C03563=1012.547,271.905,-142.723,165.559,65.313,161.899
C03564=1012.520,272.316,-142.820,165.483,65.289,161.863
C03565=1012.492,272.726,-142.918,165.407,65.263,161.827
C03566=1012.478,272.932,-142.967,165.366,65.262,161.811
C03567=1012.464,273.137,-143.018,165.328,65.252,161.794
C03568=1012.450,273.343,-143.067,165.291,65.234,161.775
C03569=1012.435,273.549,-143.117,165.257,65.209,161.756
C03570=1012.418,273.754,-143.168,165.216,65.208,161.739
C03571=1012.404,273.958,-143.220,165.178,65.197,161.722
C03572=1012.388,274.163,-143.271,165.142,65.178,161.703
C03573=1012.372,274.369,-143.324,165.099,65.180,161.687
C03574=1012.356,274.573,-143.376,165.058,65.174,161.670
C03575=1012.338,274.778,-143.429,165.021,65.161,161.652
C03576=1012.322,274.984,-143.482,164.985,65.139,161.633
C03577=1012.305,275.188,-143.536,164.946,65.130,161.616
C03578=1012.288,275.393,-143.589,164.907,65.119,161.598
C03579=1012.270,275.598,-143.644,164.868,65.109,161.580
C03580=1012.252,275.802,-143.699,164.825,65.106,161.563
C03581=1012.233,276.007,-143.754,164.788,65.094,161.546
C03582=1012.215,276.212,-143.810,164.751,65.074,161.527
C03583=1012.196,276.416,-143.866,164.709,65.071,161.510
C03584=1012.178,276.621,-143.922,164.668,65.064,161.492
C03585=1012.158,276.825,-143.978,164.631,65.048,161.474
C03586=1012.139,277.029,-144.036,164.593,65.032,161.456
C03587=1012.119,277.234,-144.094,164.552,65.025,161.439
C03588=1012.099,277.438,-144.151,164.515,65.008,161.420
C03589=1012.078,277.643,-144.210,164.471,65.007,161.403
C03590=1012.057,277.846,-144.269,164.432,64.996,161.385
C03591=1012.037,278.050,-144.327,164.395,64.977,161.367
C03592=1012.016,278.254,-144.387,164.350,64.978,161.350
C03593=1011.993,278.458,-144.448,164.307,64.973,161.332
C03594=1011.972,278.662,-144.508,164.268,64.959,161.314
C03595=1011.950,278.866,-144.568,164.233,64.936,161.295
C03596=1011.928,279.070,-144.629,164.193,64.926,161.278
C03597=1011.905,279.273,-144.691,164.153,64.915,161.260
C03598=1011.882,279.477,-144.753,164.112,64.905,161.242
C03599=1011.858,279.680,-144.815,164.067,64.904,161.224
C03600=1011.835,279.883,-144.878,164.026,64.895,161.206
C03601=1011.811,280.087,-144.941,163.989,64.876,161.188
C03602=1011.787,280.290,-145.004,163.951,64.858,161.170
C03603=1011.763,280.493,-145.069,163.905,64.859,161.152
C03604=1011.738,280.696,-145.133,163.863,64.849,161.134
C03605=1011.713,280.899,-145.198,163.825,64.831,161.116
C03606=1011.688,281.103,-145.263,163.788,64.810,161.097
C03607=1011.663,281.305,-145.328,163.744,64.803,161.079
C03608=1011.636,281.508,-145.395,163.704,64.790,161.061
C03609=1011.610,281.711,-145.461,163.662,64.778,161.042
C03610=1011.584,281.913,-145.528,163.616,64.774,161.024
C03611=1011.557,282.116,-145.596,163.574,64.761,161.005
C03612=1011.529,282.319,-145.662,163.538,64.739,160.987
C03613=1011.503,282.521,-145.731,163.495,64.728,160.968
C03614=1011.476,282.724,-145.799,163.454,64.713,160.950
C03615=1011.447,282.926,-145.868,163.410,64.703,160.931
C03616=1011.418,283.128,-145.937,163.368,64.691,160.912
C03617=1011.390,283.330,-146.007,163.326,64.677,160.894
C03618=1011.361,283.532,-146.078,163.280,64.670,160.874
C03619=1011.332,283.734,-146.148,163.238,64.655,160.856
C03620=1011.302,283.936,-146.219,163.197,64.637,160.837
C03621=1011.273,284.137,-146.291,163.151,64.631,160.818
C03622=1011.242,284.338,-146.363,163.108,64.616,160.799
C03623=1011.212,284.540,-146.435,163.070,64.595,160.780
C03624=1011.182,284.741,-146.508,163.025,64.585,160.761
C03625=1011.150,284.942,-146.581,162.982,64.568,160.741
C03626=1011.119,285.143,-146.656,162.934,64.561,160.722
C03627=1011.087,285.344,-146.730,162.892,64.544,160.703
C03628=1011.055,285.545,-146.804,162.848,64.531,160.684
C03629=1011.022,285.746,-146.879,162.800,64.525,160.664
C03630=1010.989,285.947,-146.955,162.755,64.510,160.645
C03631=1010.957,286.148,-147.030,162.717,64.486,160.626
C03632=1010.924,286.348,-147.108,162.673,64.472,160.607
C03633=1010.890,286.548,-147.184,162.629,64.455,160.587
C03634=1010.856,286.749,-147.261,162.583,64.442,160.567
C03635=1010.821,286.948,-147.340,162.537,64.428,160.547
C03636=1010.787,287.148,-147.418,162.494,64.411,160.528
C03637=1010.752,287.349,-147.497,162.441,64.405,160.507
C03638=1010.716,287.548,-147.577,162.396,64.390,160.487
C03639=1010.681,287.748,-147.655,162.357,64.364,160.468
C03640=1010.644,287.947,-147.736,162.307,64.353,160.447
C03641=1010.608,288.146,-147.817,162.257,64.344,160.427
C03642=1010.572,288.346,-147.898,162.214,64.323,160.407
C03643=1010.535,288.544,-147.979,162.174,64.295,160.388
C03644=1010.497,288.744,-148.061,162.124,64.284,160.367
C03645=1010.460,288.942,-148.144,162.080,64.263,160.347
C03646=1010.422,289.141,-148.227,162.030,64.252,160.326
C03647=1010.383,289.339,-148.311,161.979,64.239,160.305
C03648=1010.344,289.538,-148.395,161.936,64.215,160.285
C03649=1010.305,289.736,-148.479,161.891,64.194,160.264
C03650=1010.266,289.934,-148.564,161.845,64.176,160.244
C03651=1010.226,290.132,-148.651,161.795,64.160,160.223
C03652=1010.185,290.330,-148.737,161.748,64.140,160.202
C03653=1010.144,290.528,-148.823,161.698,64.124,160.181
C03654=1010.104,290.725,-148.910,161.650,64.107,160.160
C03655=1010.063,290.922,-148.998,161.604,64.085,160.140
C03656=1010.020,291.119,-149.086,161.550,64.072,160.117
C03657=1009.979,291.316,-149.175,161.505,64.049,160.097
C03658=1009.936,291.513,-149.264,161.455,64.031,160.076
C03659=1009.893,291.709,-149.354,161.403,64.014,160.054
C03660=1009.850,291.905,-149.444,161.360,63.987,160.034
C03661=1009.807,292.102,-149.534,161.307,63.969,160.012
C03662=1009.763,292.298,-149.626,161.261,63.946,159.991
C03663=1009.717,292.494,-149.718,161.204,63.933,159.968
C03664=1009.673,292.689,-149.810,161.158,63.908,159.947
C03665=1009.628,292.884,-149.904,161.102,63.893,159.925
C03666=1009.582,293.080,-149.997,161.048,63.877,159.902
C03667=1009.536,293.275,-150.091,161.002,63.850,159.881
C03668=1009.490,293.470,-150.186,160.954,63.825,159.860
C03669=1009.443,293.665,-150.280,160.905,63.802,159.839
C03670=1009.395,293.859,-150.377,160.851,63.783,159.816
C03671=1009.348,294.053,-150.473,160.801,63.760,159.794
C03672=1009.300,294.247,-150.570,160.747,63.740,159.772
C03673=1009.252,294.441,-150.668,160.694,63.718,159.749
C03674=1009.202,294.634,-150.766,160.645,63.691,159.728
C03675=1009.154,294.828,-150.865,160.587,63.674,159.704
C03676=1009.103,295.022,-150.964,160.541,63.645,159.683
C03677=1009.054,295.215,-151.064,160.482,63.627,159.660
C03678=1009.003,295.406,-151.164,160.432,63.601,159.638
C03679=1008.952,295.600,-151.265,160.380,63.576,159.616
C03680=1008.900,295.792,-151.366,160.329,63.549,159.594
C03681=1008.848,295.984,-151.469,160.271,63.530,159.570
C03682=1008.796,296.176,-151.571,160.222,63.501,159.548
C03683=1008.743,296.367,-151.675,160.159,63.483,159.523
C03684=1008.690,296.558,-151.780,160.105,63.459,159.500
C03685=1008.637,296.749,-151.884,160.061,63.424,159.480
C03686=1008.582,296.940,-151.990,160.004,63.400,159.457
C03687=1008.528,297.130,-152.095,159.950,63.375,159.434
C03688=1008.473,297.320,-152.201,159.895,63.348,159.411
C03689=1008.417,297.510,-152.309,159.839,63.323,159.388
C03690=1008.362,297.699,-152.417,159.785,63.296,159.365
C03691=1008.305,297.889,-152.526,159.728,63.270,159.342
C03692=1008.248,298.078,-152.634,159.671,63.243,159.318
C03693=1008.191,298.267,-152.744,159.622,63.210,159.296
C03694=1008.133,298.454,-152.855,159.557,63.191,159.271
C03695=1008.074,298.643,-152.966,159.506,63.158,159.249
C03696=1008.016,298.831,-153.077,159.453,63.128,159.227
C03697=1007.957,299.018,-153.190,159.391,63.104,159.202
C03698=1007.897,299.205,-153.303,159.343,63.067,159.181
C03699=1007.837,299.392,-153.416,159.288,63.037,159.158
C03700=1007.776,299.579,-153.531,159.236,63.004,159.136
C03701=1007.715,299.765,-153.646,159.173,62.979,159.111
C03702=1007.653,299.952,-153.762,159.119,62.947,159.088
C03703=1007.591,300.137,-153.877,159.069,62.911,159.067
C03704=1007.529,300.322,-153.994,159.016,62.877,159.044
C03705=1007.465,300.507,-154.112,158.956,62.848,159.020
C03706=1007.402,300.691,-154.231,158.901,62.815,158.997
C03707=1007.338,300.875,-154.350,158.845,62.782,158.974
C03708=1007.273,301.059,-154.469,158.787,62.751,158.951
C03709=1007.208,301.243,-154.590,158.732,62.717,158.928
C03710=1007.142,301.425,-154.711,158.675,62.684,158.905
C03711=1007.076,301.608,-154.833,158.617,62.651,158.881
C03712=1007.010,301.791,-154.955,158.570,62.610,158.861
C03713=1006.943,301.973,-155.079,158.508,62.579,158.837
C03714=1006.875,302.154,-155.203,158.460,62.538,158.816
C03715=1006.806,302.335,-155.327,158.397,62.508,158.791
C03716=1006.738,302.516,-155.452,158.351,62.465,158.772
C03717=1006.669,302.697,-155.578,158.293,62.430,158.748
C03718=1006.599,302.877,-155.705,158.234,62.395,158.725
C03719=1006.529,303.056,-155.832,158.183,62.355,158.704
C03720=1006.458,303.235,-155.961,158.119,62.323,158.679
C03721=1006.386,303.413,-156.089,158.065,62.284,158.657
C03722=1006.315,303.591,-156.219,158.019,62.240,158.637
C03723=1006.243,303.769,-156.349,157.967,62.199,158.616
C03724=1006.170,303.946,-156.480,157.907,62.163,158.592
C03725=1006.096,304.123,-156.611,157.854,62.123,158.571
C03726=1006.022,304.300,-156.744,157.799,62.083,158.549
C03727=1005.948,304.475,-156.877,157.743,62.044,158.527
C03728=1005.873,304.650,-157.011,157.689,62.003,158.505
C03729=1005.797,304.826,-157.146,157.635,61.962,158.484
C03730=1005.721,305.000,-157.281,157.577,61.924,158.461
C03731=1005.645,305.174,-157.416,157.536,61.875,158.444
C03732=1005.568,305.347,-157.554,157.473,61.838,158.420
C03733=1005.489,305.521,-157.691,157.431,61.789,158.402
C03734=1005.411,305.693,-157.829,157.369,61.752,158.378
C03735=1005.332,305.865,-157.968,157.326,61.702,158.360
C03736=1005.253,306.036,-158.107,157.270,61.661,158.339
C03737=1005.173,306.206,-158.248,157.216,61.619,158.317
C03738=1005.092,306.376,-158.388,157.167,61.572,158.298
C03739=1005.011,306.545,-158.531,157.107,61.532,158.275
C03740=1004.930,306.715,-158.673,157.056,61.487,158.255
C03741=1004.849,306.884,-158.817,157.015,61.437,158.238
C03742=1004.766,307.052,-158.961,156.968,61.390,158.220
C03743=1004.683,307.219,-159.105,156.912,61.346,158.198
C03744=1004.599,307.386,-159.250,156.864,61.300,158.180
C03745=1004.514,307.552,-159.396,156.812,61.255,158.160
C03746=1004.430,307.718,-159.543,156.761,61.208,158.140
C03747=1004.344,307.882,-159.690,156.711,61.161,158.121
C03748=1004.258,308.047,-159.838,156.664,61.113,158.103
C03749=1004.171,308.210,-159.988,156.609,61.069,158.083
C03750=1004.085,308.374,-160.136,156.576,61.015,158.068
C03751=1003.997,308.536,-160.287,156.513,60.973,158.046
C03752=1003.909,308.698,-160.438,156.475,60.920,158.030
C03753=1003.821,308.859,-160.590,156.422,60.874,158.011
C03754=1003.731,309.020,-160.742,156.376,60.825,157.993
C03755=1003.643,309.180,-160.895,156.338,60.772,157.978
C03756=1003.553,309.339,-161.049,156.294,60.722,157.961
C03757=1003.461,309.498,-161.203,156.240,60.676,157.942
C03758=1003.370,309.655,-161.358,156.200,60.624,157.926
C03759=1003.279,309.812,-161.514,156.145,60.578,157.907
C03760=1003.186,309.969,-161.670,156.096,60.531,157.889
C03761=1003.093,310.126,-161.827,156.071,60.473,157.878
C03762=1002.943,310.375,-162.081,156.002,60.391,157.852
C03763=1002.792,310.621,-162.337,155.930,60.312,157.826
C03764=1002.639,310.867,-162.595,155.857,60.232,157.799
C03765=1002.484,311.110,-162.853,155.787,60.151,157.774
C03766=1002.501,310.643,-162.969,145.440,63.688,154.150
C03767=1002.632,310.435,-162.749,145.501,63.818,154.157
C03768=1002.762,310.226,-162.532,145.576,63.944,154.169
C03769=1002.890,310.016,-162.315,145.657,64.070,154.183
C03770=1003.017,309.805,-162.100,145.734,64.195,154.197
C03771=1003.108,309.650,-161.944,145.769,64.292,154.198
C03772=1003.201,309.494,-161.789,145.833,64.381,154.211
C03773=1003.292,309.339,-161.634,145.905,64.468,154.228
C03774=1003.382,309.182,-161.480,145.957,64.561,154.237
C03775=1003.472,309.025,-161.327,146.027,64.648,154.253
C03776=1003.562,308.867,-161.174,146.087,64.738,154.266
C03777=1003.651,308.708,-161.023,146.140,64.831,154.275
C03778=1003.739,308.548,-160.871,146.202,64.921,154.289
C03779=1003.827,308.389,-160.720,146.273,65.008,154.306
C03780=1003.914,308.228,-160.571,146.328,65.100,154.317
C03781=1004.001,308.067,-160.422,146.411,65.183,154.340
C03782=1004.087,307.905,-160.273,146.461,65.277,154.349
C03783=1004.173,307.743,-160.126,146.534,65.362,154.369
C03784=1004.258,307.580,-159.979,146.603,65.450,154.386
C03785=1004.342,307.416,-159.833,146.672,65.535,154.404
C03786=1004.426,307.251,-159.687,146.745,65.621,154.424
C03787=1004.510,307.086,-159.543,146.816,65.706,154.444
C03788=1004.594,306.921,-159.398,146.887,65.791,154.463
C03789=1004.676,306.754,-159.254,146.965,65.874,154.486
C03790=1004.758,306.589,-159.111,147.035,65.959,154.505
C03791=1004.839,306.421,-158.970,147.097,66.047,154.521
C03792=1004.920,306.253,-158.828,147.171,66.132,154.543
C03793=1005.000,306.085,-158.687,147.258,66.209,154.571
C03794=1005.080,305.916,-158.547,147.331,66.294,154.592
C03795=1005.159,305.746,-158.408,147.412,66.374,154.618
C03796=1005.238,305.577,-158.270,147.494,66.453,154.644
C03797=1005.316,305.406,-158.131,147.559,66.540,154.663
C03798=1005.394,305.235,-157.994,147.653,66.615,154.695
C03799=1005.471,305.063,-157.858,147.719,66.700,154.715
C03800=1005.548,304.892,-157.722,147.811,66.774,154.746
C03801=1005.623,304.719,-157.588,147.878,66.859,154.767
C03802=1005.699,304.546,-157.454,147.965,66.935,154.797
C03803=1005.774,304.372,-157.320,148.049,67.012,154.826
C03804=1005.848,304.198,-157.187,148.132,67.088,154.855
C03805=1005.923,304.024,-157.055,148.219,67.164,154.885
C03806=1005.995,303.849,-156.924,148.305,67.238,154.916
C03807=1006.068,303.674,-156.793,148.389,67.314,154.946
C03808=1006.141,303.497,-156.663,148.482,67.385,154.980
C03809=1006.213,303.321,-156.533,148.565,67.461,155.010
C03810=1006.284,303.144,-156.405,148.642,67.538,155.038
C03811=1006.355,302.966,-156.277,148.728,67.612,155.069
C03812=1006.425,302.789,-156.149,148.828,67.678,155.108
C03813=1006.494,302.611,-156.023,148.913,67.752,155.140
C03814=1006.564,302.432,-155.898,149.007,67.820,155.176
C03815=1006.633,302.254,-155.772,149.102,67.888,155.213
C03816=1006.700,302.075,-155.648,149.179,67.965,155.242
C03817=1006.768,301.895,-155.524,149.281,68.028,155.283
C03818=1006.836,301.714,-155.401,149.363,68.101,155.314
C03819=1006.902,301.534,-155.278,149.463,68.164,155.355
C03820=1006.968,301.352,-155.158,149.544,68.237,155.387
C03821=1007.034,301.171,-155.036,149.640,68.301,155.426
C03822=1007.099,300.989,-154.916,149.737,68.366,155.466
C03823=1007.163,300.807,-154.797,149.829,68.432,155.503
C03824=1007.228,300.625,-154.678,149.927,68.494,155.544
C03825=1007.291,300.443,-154.559,150.020,68.558,155.583
C03826=1007.354,300.259,-154.442,150.116,68.620,155.623
C03827=1007.417,300.076,-154.325,150.216,68.680,155.666
C03828=1007.479,299.892,-154.209,150.309,68.744,155.705
C03829=1007.541,299.707,-154.093,150.398,68.809,155.743
C03830=1007.602,299.522,-153.979,150.492,68.871,155.783
C03831=1007.663,299.338,-153.864,150.599,68.924,155.830
C03832=1007.723,299.153,-153.751,150.690,68.986,155.869
C03833=1007.782,298.967,-153.638,150.787,69.046,155.912
C03834=1007.842,298.781,-153.526,150.875,69.110,155.950
C03835=1007.901,298.595,-153.414,150.980,69.162,155.997
C03836=1007.959,298.407,-153.304,151.076,69.221,156.040
C03837=1008.016,298.221,-153.193,151.170,69.280,156.081
C03838=1008.074,298.034,-153.083,151.280,69.328,156.132
C03839=1008.131,297.846,-152.975,151.372,69.388,156.173
C03840=1008.187,297.658,-152.865,151.474,69.440,156.220
C03841=1008.244,297.471,-152.758,151.575,69.493,156.266
C03842=1008.299,297.282,-152.651,151.672,69.546,156.310
C03843=1008.354,297.093,-152.544,151.775,69.597,156.358
C03844=1008.409,296.905,-152.438,151.874,69.650,156.404
C03845=1008.463,296.716,-152.333,151.974,69.700,156.450
C03846=1008.517,296.526,-152.228,152.078,69.749,156.499
C03847=1008.569,296.336,-152.124,152.162,69.809,156.538
C03848=1008.622,296.146,-152.022,152.262,69.859,156.586
C03849=1008.674,295.956,-151.918,152.373,69.900,156.638
C03850=1008.727,295.765,-151.816,152.468,69.953,156.684
C03851=1008.778,295.575,-151.713,152.575,69.996,156.735
C03852=1008.830,295.384,-151.613,152.670,70.046,156.780
C03853=1008.880,295.193,-151.513,152.767,70.096,156.827
C03854=1008.930,295.001,-151.413,152.866,70.144,156.875
C03855=1008.980,294.809,-151.313,152.972,70.186,156.926
C03856=1009.029,294.617,-151.216,153.064,70.237,156.971
C03857=1009.079,294.426,-151.117,153.172,70.277,157.024
C03858=1009.127,294.233,-151.020,153.265,70.327,157.070
C03859=1009.175,294.040,-150.922,153.366,70.369,157.119
C03860=1009.223,293.847,-150.826,153.467,70.411,157.169
C03861=1009.270,293.654,-150.730,153.565,70.456,157.218
C03862=1009.317,293.461,-150.635,153.667,70.497,157.269
C03863=1009.364,293.267,-150.540,153.765,70.540,157.317
C03864=1009.409,293.074,-150.446,153.859,70.586,157.365
C03865=1009.456,292.879,-150.353,153.950,70.634,157.411
C03866=1009.501,292.685,-150.260,154.054,70.670,157.463
C03867=1009.546,292.491,-150.167,154.161,70.706,157.517
C03868=1009.591,292.297,-150.075,154.254,70.750,157.564
C03869=1009.634,292.103,-149.984,154.361,70.783,157.618
C03870=1009.678,291.907,-149.893,154.456,70.826,157.667
C03871=1009.722,291.712,-149.802,154.556,70.863,157.718
C03872=1009.764,291.517,-149.713,154.646,70.909,157.764
C03873=1009.808,291.322,-149.624,154.747,70.944,157.816
C03874=1009.850,291.126,-149.535,154.847,70.981,157.868
C03875=1009.891,290.929,-149.447,154.939,71.022,157.916
C03876=1009.933,290.735,-149.358,155.044,71.054,157.970
C03877=1009.974,290.538,-149.272,155.138,71.094,158.019
C03878=1010.015,290.342,-149.186,155.235,71.129,158.069
C03879=1010.055,290.145,-149.099,155.335,71.162,158.121
C03880=1010.095,289.949,-149.013,155.429,71.200,158.171
C03881=1010.134,289.751,-148.928,155.529,71.233,158.223
C03882=1010.174,289.555,-148.843,155.624,71.269,158.273
C03883=1010.213,289.357,-148.760,155.718,71.307,158.323
C03884=1010.251,289.160,-148.676,155.807,71.347,158.371
C03885=1010.290,288.963,-148.593,155.908,71.376,158.424
C03886=1010.327,288.765,-148.510,156.011,71.405,158.478
C03887=1010.365,288.567,-148.428,156.103,71.442,158.527
C03888=1010.402,288.369,-148.346,156.204,71.468,158.581
C03889=1010.439,288.171,-148.265,156.288,71.512,158.627
C03890=1010.475,287.973,-148.185,156.380,71.548,158.677
C03891=1010.511,287.775,-148.104,156.482,71.574,158.731
C03892=1010.547,287.577,-148.024,156.581,71.600,158.784
C03893=1010.583,287.378,-147.945,156.667,71.641,158.831
C03894=1010.618,287.179,-147.865,156.763,71.672,158.883
C03895=1010.653,286.981,-147.787,156.868,71.692,158.938
C03896=1010.687,286.781,-147.709,156.961,71.724,158.989
C03897=1010.722,286.582,-147.632,157.055,71.753,159.040
C03898=1010.756,286.383,-147.554,157.151,71.779,159.093
C03899=1010.789,286.184,-147.478,157.244,71.810,159.143
C03900=1010.822,285.984,-147.402,157.339,71.839,159.195
C03901=1010.855,285.785,-147.326,157.423,71.877,159.242
C03902=1010.887,285.585,-147.252,157.517,71.906,159.294
C03903=1010.919,285.385,-147.176,157.617,71.925,159.348
C03904=1010.951,285.186,-147.102,157.711,71.953,159.399
C03905=1010.982,284.985,-147.029,157.802,71.983,159.450
C03906=1011.014,284.786,-146.955,157.902,72.002,159.504
C03907=1011.045,284.585,-146.881,157.993,72.033,159.555
C03908=1011.075,284.385,-146.809,158.088,72.056,159.607
C03909=1011.105,284.184,-146.737,158.174,72.090,159.656
C03910=1011.135,283.984,-146.666,158.267,72.118,159.708
C03911=1011.165,283.783,-146.594,158.365,72.136,159.761
C03912=1011.194,283.582,-146.523,158.455,72.167,159.812
C03913=1011.224,283.381,-146.453,158.545,72.195,159.863
C03914=1011.252,283.181,-146.384,158.643,72.214,159.917
C03915=1011.281,282.979,-146.314,158.735,72.240,159.968
C03916=1011.309,282.777,-146.245,158.827,72.264,160.020
C03917=1011.337,282.577,-146.176,158.923,72.286,160.073
C03918=1011.364,282.376,-146.108,159.014,72.313,160.125
C03919=1011.392,282.174,-146.040,159.107,72.336,160.177
C03920=1011.418,281.972,-145.974,159.191,72.370,160.226
C03921=1011.445,281.771,-145.906,159.282,72.394,160.278
C03922=1011.471,281.569,-145.839,159.381,72.410,160.332
C03923=1011.497,281.367,-145.773,159.472,72.432,160.384
C03924=1011.523,281.165,-145.707,159.561,72.458,160.435
C03925=1011.548,280.963,-145.642,159.657,72.475,160.488
C03926=1011.574,280.761,-145.577,159.742,72.508,160.538
C03927=1011.598,280.559,-145.513,159.830,72.537,160.590
C03928=1011.622,280.357,-145.449,159.923,72.556,160.642
C03929=1011.648,280.155,-145.385,160.020,72.566,160.695
C03930=1011.672,279.952,-145.322,160.106,72.595,160.746
C03931=1011.695,279.750,-145.260,160.192,72.623,160.796
C03932=1011.719,279.547,-145.196,160.284,72.643,160.848
C03933=1011.742,279.345,-145.134,160.380,72.654,160.902
C03934=1011.765,279.142,-145.073,160.471,72.674,160.954
C03935=1011.787,278.939,-145.011,160.561,72.696,161.006
C03936=1011.809,278.736,-144.951,160.653,72.716,161.058
C03937=1011.831,278.534,-144.891,160.737,72.748,161.109
C03938=1011.853,278.330,-144.830,160.827,72.772,161.161
C03939=1011.875,278.128,-144.770,160.920,72.787,161.214
C03940=1011.896,277.925,-144.711,161.016,72.795,161.267
C03941=1011.916,277.721,-144.652,161.104,72.824,161.320
C03942=1011.937,277.519,-144.593,161.194,72.844,161.372
C03943=1011.958,277.315,-144.535,161.289,72.854,161.425
C03944=1011.978,277.112,-144.478,161.376,72.880,161.477
C03945=1011.998,276.908,-144.421,161.468,72.898,161.530
C03946=1012.017,276.705,-144.364,161.556,72.922,161.583
C03947=1012.036,276.501,-144.307,161.644,72.947,161.635
C03948=1012.055,276.298,-144.251,161.737,72.963,161.688
C03949=1012.074,276.094,-144.196,161.830,72.974,161.741
C03950=1012.092,275.890,-144.140,161.917,73.004,161.794
C03951=1012.110,275.687,-144.085,162.007,73.024,161.847
C03952=1012.128,275.483,-144.031,162.100,73.036,161.900
C03953=1012.163,275.075,-143.923,162.281,73.074,162.007
C03954=1012.196,274.667,-143.816,162.459,73.122,162.114
C03955=1012.229,274.259,-143.711,162.640,73.157,162.220
C03956=1012.261,273.850,-143.607,162.821,73.190,162.326
C03957=1012.291,273.441,-143.506,163.004,73.218,162.433
C03958=1012.320,273.033,-143.406,163.179,73.277,162.542
C03959=1012.349,272.624,-143.307,163.361,73.302,162.648
C03960=1012.376,272.215,-143.210,163.541,73.345,162.757
C03961=1012.403,271.805,-143.114,163.720,73.382,162.865
C03962=1012.429,271.396,-143.019,163.904,73.408,162.973
C03963=1012.453,270.986,-142.926,164.083,73.457,163.084
C03964=1012.476,270.576,-142.835,164.268,73.472,163.190
C03965=1012.498,270.166,-142.745,164.448,73.516,163.301
C03966=1012.520,269.756,-142.656,164.629,73.543,163.409
C03967=1012.539,269.345,-142.570,164.811,73.603,163.526
C03968=1012.558,268.935,-142.484,164.993,73.628,163.635
C03969=1012.576,268.525,-142.400,165.176,73.659,163.745
C03970=1012.593,268.113,-142.318,165.359,73.707,163.861
C03971=1012.610,267.702,-142.236,165.542,73.721,163.967
C03972=1012.625,267.291,-142.157,165.725,73.766,164.083
C03973=1012.638,266.880,-142.079,165.909,73.798,164.196
C03974=1012.651,266.468,-142.001,166.092,73.823,164.306
C03975=1012.664,266.057,-141.925,166.275,73.857,164.419
C03976=1012.674,265.646,-141.852,166.460,73.903,164.537
C03977=1012.684,265.234,-141.780,166.647,73.945,164.656
C03978=1012.694,264.822,-141.708,166.828,73.953,164.761
C03979=1012.701,264.409,-141.640,167.017,74.010,164.886
C03980=1012.709,263.997,-141.571,167.202,74.042,165.001
C03981=1012.714,263.585,-141.504,167.386,74.060,165.112
C03982=1012.719,263.173,-141.439,167.573,74.109,165.235
C03983=1012.724,262.760,-141.374,167.755,74.124,165.344
C03984=1012.727,262.347,-141.313,167.944,74.166,165.466
///RCONF 0,0,0,0,1,0,0,0,0,0,0,0,0,0,0,0,0,0,0,0,0,0,0,0
C03985=1012.728,261.935,-141.252,168.129,74.189,165.580
C03986=1012.730,261.522,-141.193,168.325,74.250,165.712
C03987=1012.730,261.109,-141.135,168.510,74.275,165.828
C03988=1012.729,260.697,-141.078,168.696,74.303,165.945
C03989=1012.727,260.283,-141.024,168.890,74.352,166.074
C03990=1012.724,259.870,-140.969,169.072,74.367,166.185
C03991=1012.710,258.621,-140.814,169.635,74.457,166.544
C03992=1012.706,258.376,-140.785,169.634,74.467,166.547
C03993=1012.703,258.131,-140.756,169.632,74.475,166.549
C03994=1012.699,257.886,-140.727,169.630,74.484,166.552
C03995=1012.695,257.640,-140.698,169.627,74.493,166.553
C03996=1012.692,257.395,-140.669,169.625,74.501,166.555
C03997=1012.688,257.150,-140.640,169.624,74.509,166.557
C03998=1012.684,256.904,-140.611,169.622,74.517,166.559
C03999=1012.681,256.659,-140.582,169.620,74.526,166.561
C04000=1012.678,256.414,-140.553,169.618,74.534,166.562
C04001=1012.674,256.169,-140.524,169.614,74.541,166.563
C04002=1012.670,255.924,-140.495,169.612,74.549,166.565
C04003=1012.667,255.679,-140.466,169.611,74.559,166.568
C04004=1012.663,255.432,-140.438,169.608,74.567,166.569
C04005=1012.660,255.187,-140.409,169.607,74.577,166.572
C04006=1012.656,254.942,-140.380,169.605,74.585,166.574
C04007=1012.653,254.698,-140.351,169.602,74.594,166.575
C04008=1012.649,254.452,-140.322,169.600,74.602,166.577
C04009=1012.646,254.206,-140.294,169.598,74.610,166.579
C04010=1012.642,253.961,-140.265,169.596,74.618,166.581
C04011=1012.639,253.716,-140.236,169.594,74.626,166.583
C04012=1012.635,253.471,-140.207,169.592,74.634,166.584
C04013=1012.632,253.225,-140.178,169.591,74.642,166.586
C04014=1012.628,252.980,-140.149,169.587,74.651,166.588
C04015=1012.625,252.735,-140.121,169.586,74.661,166.591
C04016=1012.621,252.489,-140.092,169.583,74.669,166.592
C04017=1012.618,252.244,-140.063,169.583,74.678,166.595
C04018=1012.614,251.999,-140.034,169.580,74.687,166.597
C04019=1012.611,251.753,-140.006,169.578,74.695,166.599
C04020=1012.608,251.508,-139.977,169.577,74.703,166.601
C04021=1012.604,251.263,-139.948,169.575,74.711,166.602
C04022=1012.601,251.017,-139.920,169.573,74.720,166.604
C04023=1012.597,250.772,-139.891,169.571,74.728,166.606
C04024=1012.594,250.526,-139.863,169.568,74.736,166.608
C04025=1012.590,250.282,-139.834,169.567,74.746,166.611
C04026=1012.586,250.037,-139.806,169.566,74.755,166.613
C04027=1012.583,249.791,-139.777,169.564,74.764,166.615
C04028=1012.579,249.545,-139.748,169.563,74.773,166.618
C04029=1012.576,249.300,-139.720,169.561,74.781,166.620
C04030=1012.573,249.055,-139.691,169.558,74.790,166.621
C04031=1012.570,248.809,-139.663,169.556,74.798,166.623
C04032=1012.566,248.564,-139.634,169.554,74.806,166.625
C04033=1012.563,248.319,-139.606,169.553,74.814,166.627
C04034=1012.560,248.073,-139.578,169.551,74.822,166.629
C04035=1012.557,247.828,-139.549,169.550,74.832,166.632
C04036=1012.554,247.583,-139.521,169.549,74.841,166.635
C04037=1012.549,247.337,-139.491,169.546,74.850,166.636
C04038=1012.546,247.091,-139.463,169.546,74.859,166.640
C04039=1012.543,246.846,-139.435,169.543,74.868,166.641
C04040=1012.540,246.601,-139.406,169.543,74.877,166.644
C04041=1012.537,246.355,-139.378,169.540,74.885,166.646
C04042=1012.534,246.110,-139.350,169.538,74.894,166.648
C04043=1012.530,245.865,-139.321,169.536,74.902,166.650
C04044=1012.526,245.619,-139.293,169.534,74.910,166.652
C04045=1012.523,245.374,-139.265,169.533,74.918,166.654
C04046=1012.520,245.129,-139.236,169.532,74.928,166.657
C04047=1012.517,244.883,-139.208,169.531,74.937,166.659
C04048=1012.514,244.637,-139.180,169.530,74.947,166.662
C04049=1012.510,244.392,-139.152,169.527,74.955,166.664
C04050=1012.507,244.147,-139.123,169.526,74.965,166.667
C04051=1012.504,243.901,-139.095,169.524,74.973,166.669
C04052=1012.501,243.656,-139.067,169.524,74.982,166.672
C04053=1012.498,243.410,-139.038,169.521,74.991,166.673
C04054=1012.495,243.165,-139.010,169.519,74.999,166.675
C04055=1012.491,242.920,-138.981,169.517,75.007,166.677
C04056=1012.488,242.674,-138.953,169.516,75.016,166.680
C04057=1012.485,242.428,-138.925,169.513,75.025,166.682
C04058=1012.482,242.183,-138.897,169.512,75.035,166.685
C04059=1012.478,241.937,-138.869,169.513,75.044,166.688
C04060=1012.475,241.692,-138.841,169.512,75.053,166.691
C04061=1012.472,241.446,-138.813,169.509,75.062,166.693
///RCONF 0,0,0,0,0,0,0,0,0,0,0,0,0,0,0,0,0,0,0,0,0,0,0,0
C04062=1012.469,241.201,-138.785,169.509,75.071,166.696
C04063=1012.466,240.955,-138.757,169.506,75.080,166.697
C04064=1012.463,240.711,-138.728,169.504,75.088,166.699
C04065=1012.460,240.465,-138.700,169.505,75.097,166.703
C04066=1012.456,240.220,-138.672,169.503,75.105,166.705
C04067=1012.453,239.974,-138.644,169.502,75.114,166.708
C04068=1012.450,239.728,-138.615,169.501,75.124,166.711
C04069=1012.447,239.483,-138.587,169.498,75.133,166.712
C04070=1012.444,239.237,-138.559,169.497,75.142,166.715
C04071=1012.441,238.992,-138.531,169.496,75.152,166.718
C04072=1012.438,238.745,-138.503,169.496,75.161,166.722
C04073=1012.434,238.500,-138.476,169.493,75.169,166.723
C04074=1012.432,238.255,-138.448,169.494,75.178,166.727
C04075=1012.429,238.010,-138.420,169.491,75.187,166.728
C04076=1012.425,237.764,-138.392,169.489,75.195,166.730
C04077=1012.422,237.518,-138.364,169.487,75.203,166.732
C04078=1012.419,237.273,-138.335,169.486,75.213,166.735
C04079=1012.416,237.027,-138.307,169.488,75.223,166.739
C04080=1012.414,236.782,-138.279,169.485,75.232,166.741
C04081=1012.411,236.536,-138.252,169.484,75.241,166.744
C04082=1012.408,236.291,-138.224,169.483,75.251,166.747
C04083=1012.405,236.045,-138.196,169.482,75.261,166.750
C04084=1012.401,235.799,-138.168,169.480,75.269,166.752
C04085=1012.398,235.554,-138.139,169.479,75.278,166.755
C04086=1012.396,235.308,-138.112,169.478,75.286,166.757
C04087=1012.393,235.063,-138.084,169.478,75.295,166.761
C04088=1012.389,234.817,-138.057,169.475,75.304,166.762
C04089=1012.386,234.572,-138.028,169.474,75.314,166.765
C04090=1012.383,234.325,-138.001,169.473,75.323,166.768
C04091=1012.381,234.081,-137.973,169.473,75.333,166.771
C04092=1012.378,233.835,-137.945,169.472,75.342,166.774
C04093=1012.375,233.589,-137.917,169.471,75.352,166.777
C04094=1012.372,233.343,-137.889,169.471,75.361,166.781
C04095=1012.369,233.098,-137.862,169.468,75.369,166.782
C04096=1012.366,232.853,-137.833,169.469,75.378,166.786
C04097=1012.363,232.606,-137.806,169.468,75.388,166.789
C04098=1012.360,232.361,-137.778,169.466,75.396,166.791
C04099=1012.358,232.115,-137.751,169.465,75.406,166.794
C04100=1012.355,231.870,-137.722,169.465,75.415,166.797
C04101=1012.351,231.624,-137.695,169.464,75.425,166.800
C04102=1012.349,231.379,-137.668,169.463,75.434,166.803
C04103=1012.346,231.133,-137.640,169.462,75.444,166.806
C04104=1012.343,230.887,-137.612,169.461,75.453,166.809
C04105=1012.340,230.642,-137.584,169.461,75.463,166.812
C04106=1012.338,230.396,-137.557,169.459,75.471,166.814
C04107=1012.334,230.150,-137.529,169.458,75.481,166.817
C04108=1012.332,229.904,-137.501,169.459,75.490,166.821
C04109=1012.329,229.659,-137.474,169.457,75.498,166.823
C04110=1012.326,229.413,-137.446,169.455,75.508,166.826
C04111=1012.323,229.167,-137.418,169.456,75.518,166.830
C04112=1012.321,228.922,-137.391,169.456,75.528,166.833
C04113=1012.318,228.676,-137.363,169.455,75.537,166.836
C04114=1012.315,228.430,-137.335,169.454,75.547,166.840
C04115=1012.313,228.185,-137.307,169.453,75.556,166.843
C04116=1012.309,227.939,-137.281,169.454,75.565,166.846
C04117=1012.306,227.694,-137.252,169.451,75.574,166.848
C04118=1012.304,227.448,-137.225,169.450,75.584,166.851
C04119=1012.301,227.202,-137.198,169.451,75.593,166.855
C04120=1012.298,226.956,-137.170,169.448,75.601,166.856
C04121=1012.296,226.711,-137.143,169.449,75.612,166.861
C04122=1012.293,226.465,-137.115,169.449,75.621,166.864
C04123=1012.290,226.220,-137.087,169.448,75.631,166.867
C04124=1012.287,225.974,-137.060,169.447,75.640,166.870
C04125=1012.285,225.727,-137.032,169.446,75.650,166.873
C04126=1012.282,225.482,-137.005,169.446,75.660,166.877
C04127=1012.279,225.236,-136.977,169.445,75.669,166.880
C04128=1012.277,224.991,-136.950,169.446,75.678,166.883
C04129=1012.274,224.745,-136.922,169.445,75.688,166.887
C04130=1012.271,224.499,-136.894,169.443,75.696,166.889
C04131=1012.269,224.253,-136.867,169.443,75.705,166.892
C04132=1012.265,224.007,-136.840,169.443,75.716,166.896
C04133=1012.263,223.762,-136.813,169.442,75.726,166.899
C04134=1012.260,223.516,-136.785,169.442,75.736,166.902
C04135=1012.258,223.271,-136.758,169.443,75.746,166.907
C04136=1012.255,223.025,-136.731,169.442,75.755,166.910
C04137=1012.252,222.778,-136.703,169.442,75.765,166.913
C04138=1012.250,222.533,-136.676,169.442,75.774,166.917
C04139=1012.247,222.287,-136.649,169.440,75.783,166.919
C04140=1012.245,222.042,-136.621,169.439,75.792,166.922
C04141=1012.242,221.796,-136.593,169.440,75.801,166.926
C04142=1012.240,221.550,-136.566,169.439,75.811,166.929
C04143=1012.237,221.304,-136.539,169.438,75.820,166.932
C04144=1012.235,221.058,-136.512,169.438,75.830,166.935
C04145=1012.232,220.812,-136.484,169.437,75.840,166.939
C04146=1012.230,220.567,-136.457,169.439,75.850,166.943
C04147=1012.227,220.317,-136.430,169.438,75.859,166.947
C04148=1012.224,220.057,-136.400,169.440,75.870,166.951
C04149=1012.221,219.785,-136.371,169.440,75.881,166.956
C04150=1012.218,219.503,-136.339,169.438,75.891,166.958
C04151=1012.215,219.208,-136.306,169.437,75.903,166.962
C04152=1012.212,218.903,-136.273,169.438,75.915,166.968
C04153=1012.210,218.608,-136.240,169.437,75.927,166.971
C04154=1012.206,218.314,-136.207,169.434,75.938,166.974
C04155=1012.204,218.025,-136.175,169.433,75.949,166.978
C04156=1012.201,217.744,-136.144,169.434,75.960,166.982
C04157=1012.198,217.479,-136.115,169.434,75.971,166.986
C04158=1012.195,217.220,-136.086,169.436,75.981,166.991
C04159=1012.193,216.965,-136.058,169.436,75.992,166.995
C04160=1012.190,216.716,-136.031,169.436,76.002,166.999
C04161=1012.188,216.470,-136.004,169.435,76.012,167.002
C04162=1012.185,216.225,-135.977,169.435,76.021,167.005
C04163=1012.183,215.979,-135.950,169.436,76.032,167.010
C04164=1012.180,215.734,-135.923,169.436,76.041,167.014
C04165=1012.178,215.489,-135.896,169.435,76.051,167.017
C04166=1012.176,215.244,-135.868,169.435,76.060,167.020
C04167=1012.173,214.998,-135.841,169.436,76.071,167.025
C04168=1012.170,214.753,-135.815,169.436,76.080,167.028
C04169=1012.168,214.509,-135.787,169.436,76.090,167.032
C04170=1012.166,214.264,-135.761,169.437,76.100,167.037
C04171=1012.164,214.019,-135.733,169.437,76.110,167.040
C04172=1012.161,213.775,-135.707,169.436,76.119,167.043
C04173=1012.159,213.531,-135.680,169.436,76.129,167.047
C04174=1012.156,213.287,-135.654,169.438,76.139,167.052
C04175=1012.155,213.044,-135.626,169.437,76.149,167.055
C04176=1012.152,212.800,-135.600,169.437,76.159,167.059
C04177=1012.150,212.557,-135.573,169.439,76.169,167.064
C04178=1012.147,212.313,-135.546,169.438,76.178,167.067
C04179=1012.145,212.070,-135.519,169.438,76.188,167.070
C04180=1012.142,211.827,-135.493,169.440,76.198,167.075
C04181=1012.140,211.584,-135.467,169.439,76.208,167.079
C04182=1012.138,211.342,-135.440,169.439,76.218,167.082
C04183=1012.136,211.099,-135.413,169.441,76.228,167.087
C04184=1012.134,210.856,-135.387,169.440,76.238,167.091
C04185=1012.131,210.614,-135.360,169.440,76.247,167.094
C04186=1012.129,210.371,-135.334,169.442,76.258,167.099
C04187=1012.127,210.128,-135.307,169.441,76.267,167.102
C04188=1012.124,209.887,-135.281,169.441,76.277,167.106
C04189=1012.122,209.644,-135.254,169.443,76.287,167.111
C04190=1012.120,209.401,-135.227,169.442,76.297,167.114
C04191=1012.118,209.159,-135.201,169.444,76.307,167.119
C04192=1012.115,208.917,-135.174,169.444,76.317,167.123
C04193=1012.113,208.673,-135.148,169.444,76.326,167.126
C04194=1012.111,208.431,-135.122,169.446,76.337,167.131
C04195=1012.109,208.189,-135.095,169.445,76.346,167.135
C04196=1012.107,207.946,-135.068,169.447,76.357,167.140
C04197=1012.105,207.703,-135.042,169.447,76.366,167.144
C04198=1012.102,207.461,-135.016,169.449,76.377,167.149
C04199=1012.100,207.218,-134.989,169.448,76.386,167.152
C04200=1012.098,206.975,-134.963,169.448,76.396,167.156
C04201=1012.096,206.732,-134.936,169.450,76.406,167.161
C04202=1012.094,206.488,-134.910,169.450,76.416,167.164
C04203=1012.091,206.245,-134.883,169.452,76.426,167.169
C04204=1012.089,206.001,-134.857,169.450,76.436,167.172
C04205=1012.087,205.758,-134.831,169.452,76.447,167.178
C04206=1012.085,205.514,-134.804,169.452,76.456,167.181
C04207=1012.083,205.270,-134.777,169.454,76.467,167.186
C04208=1012.081,205.026,-134.751,169.454,76.476,167.190
C04209=1012.078,204.782,-134.724,169.456,76.487,167.195
C04210=1012.077,204.537,-134.697,169.456,76.496,167.199
C04211=1012.074,204.293,-134.671,169.458,76.507,167.204
C04212=1012.072,204.049,-134.645,169.458,76.518,167.209
C04213=1012.070,203.806,-134.618,169.458,76.527,167.212
C04214=1012.068,203.559,-134.591,169.460,76.538,167.217
C04215=1012.062,202.309,-134.455,168.133,76.467,166.359
C04216=1012.063,202.091,-134.431,168.134,76.476,166.363
C04217=1012.063,201.885,-134.408,168.136,76.486,166.368
C04218=1012.062,201.469,-134.363,168.137,76.504,166.374
C04219=1012.064,201.252,-134.340,168.139,76.514,166.379
C04220=1012.063,201.029,-134.317,168.138,76.523,166.382
C04221=1012.063,200.790,-134.291,168.139,76.534,166.386
C04222=1012.063,200.535,-134.263,168.142,76.545,166.392
C04223=1012.063,200.281,-134.235,168.142,76.556,166.396
C04224=1012.064,200.039,-134.209,168.143,76.566,166.401
C04225=1012.063,199.807,-134.184,168.145,76.577,166.405
C04226=1012.063,199.578,-134.159,168.146,76.587,166.409
C04227=1012.064,199.335,-134.134,168.147,76.598,166.414
C04228=1012.064,198.945,-134.092,168.150,76.614,166.422
C04229=1012.064,198.553,-134.050,168.152,76.632,166.429
C04230=1012.064,198.306,-134.023,168.152,76.643,166.433
C04231=1012.064,198.070,-133.998,168.154,76.653,166.438
C04232=1012.065,197.834,-133.972,168.155,76.663,166.442
C04233=1012.065,197.598,-133.947,168.156,76.674,166.446
C04234=1012.065,197.362,-133.922,168.159,76.684,166.452
C04235=1012.066,197.126,-133.897,168.160,76.694,166.456
C04236=1012.065,196.890,-133.871,168.161,76.704,166.461
C04237=1012.065,196.654,-133.846,168.163,76.715,166.465
C04238=1012.066,196.418,-133.820,168.165,76.725,166.470
C04239=1012.065,196.182,-133.796,168.164,76.734,166.473
C04240=1012.066,195.946,-133.770,168.166,76.745,166.478
C04241=1012.066,195.710,-133.745,168.171,76.755,166.484
C04242=1012.066,195.475,-133.720,168.172,76.766,166.489
C04243=1012.067,195.239,-133.694,168.173,76.776,166.493
C04244=1012.066,195.002,-133.668,168.175,76.786,166.498
C04245=1012.066,194.766,-133.644,168.176,76.797,166.503
C04246=1012.067,194.530,-133.618,168.177,76.806,166.506
C04247=1012.067,194.294,-133.593,168.178,76.816,166.511
C04248=1012.067,194.059,-133.568,168.181,76.826,166.516
C04249=1012.067,193.823,-133.542,168.180,76.836,166.519
C04250=1012.068,193.587,-133.517,168.185,76.846,166.526
C04251=1012.068,193.351,-133.492,168.186,76.856,166.530
C04252=1012.068,193.115,-133.467,168.188,76.867,166.535
C04253=1012.069,192.879,-133.441,168.189,76.877,166.540
C04254=1012.068,192.644,-133.416,168.192,76.887,166.545
C04255=1012.069,192.407,-133.392,168.193,76.897,166.549
C04256=1012.070,192.171,-133.366,168.194,76.906,166.553
C04257=1012.069,191.935,-133.341,168.195,76.917,166.558
C04258=1012.069,191.699,-133.315,168.198,76.927,166.563
C04259=1012.070,191.463,-133.290,168.199,76.936,166.567
C04260=1012.069,191.227,-133.265,168.200,76.946,166.571
C04261=1012.070,190.991,-133.240,168.202,76.957,166.576
C04262=1012.070,190.755,-133.215,168.203,76.967,166.581
C04263=1012.070,190.519,-133.190,168.206,76.977,166.586
C04264=1012.071,190.283,-133.165,168.208,76.987,166.591
C04265=1012.071,190.047,-133.140,168.211,76.997,166.596
C04266=1012.071,189.811,-133.114,168.212,77.007,166.601
C04267=1012.072,189.576,-133.089,168.215,77.017,166.606
C04268=1012.072,189.340,-133.064,168.216,77.026,166.610
C04269=1012.073,189.104,-133.040,168.219,77.036,166.615
C04270=1012.073,188.868,-133.014,168.220,77.046,166.620
C04271=1012.073,188.632,-132.989,168.222,77.057,166.625
C04272=1012.073,188.396,-132.964,168.225,77.066,166.630
C04273=1012.073,188.161,-132.939,168.227,77.077,166.635
C04274=1012.074,187.924,-132.914,168.230,77.087,166.640
C04275=1012.074,187.688,-132.889,168.231,77.097,166.645
C04276=1012.074,187.452,-132.864,168.232,77.106,166.649
C04277=1012.075,187.216,-132.838,168.235,77.116,166.654
C04278=1012.074,186.981,-132.814,168.238,77.126,166.660
C04279=1012.075,186.744,-132.789,168.239,77.135,166.663
C04280=1012.076,186.508,-132.763,168.240,77.145,166.668
C04281=1012.076,186.273,-132.739,168.242,77.156,166.673
C04282=1012.076,186.037,-132.713,168.245,77.165,166.678
C04283=1012.076,185.801,-132.689,168.247,77.176,166.683
C04284=1012.077,185.565,-132.664,168.250,77.186,166.689
C04285=1012.077,185.329,-132.638,168.253,77.195,166.694
C04286=1012.078,184.951,-132.599,168.256,77.211,166.702
C04287=1012.078,184.622,-132.564,168.260,77.224,166.709
C04288=1012.079,184.386,-132.539,168.261,77.233,166.713
C04289=1012.078,184.150,-132.514,168.263,77.243,166.718
C04290=1012.079,183.914,-132.489,168.266,77.253,166.723
C04291=1012.080,183.678,-132.464,168.268,77.264,166.728
C04292=1012.079,183.442,-132.439,168.271,77.273,166.734
C04293=1012.081,183.206,-132.414,168.274,77.283,166.740
C04294=1012.081,182.970,-132.390,168.277,77.293,166.745
C04295=1012.081,182.734,-132.364,168.278,77.302,166.749
C04296=1012.081,182.499,-132.339,168.281,77.312,166.755
C04297=1012.082,182.262,-132.315,168.284,77.322,166.760
C04298=1012.083,182.027,-132.289,168.285,77.331,166.764
C04299=1012.082,181.791,-132.265,168.287,77.341,166.769
C04300=1012.083,181.555,-132.240,168.290,77.351,166.775
C04301=1012.083,181.319,-132.215,168.294,77.361,166.780
C04302=1012.084,181.084,-132.190,168.296,77.371,166.785
C04303=1012.084,180.848,-132.166,168.299,77.381,166.791
C04304=1012.084,180.612,-132.140,168.300,77.390,166.795
C04305=1012.084,180.376,-132.115,168.303,77.400,166.801
C04306=1012.086,180.140,-132.091,168.307,77.409,166.806
C04307=1012.085,179.904,-132.066,168.309,77.418,166.811
C04308=1012.086,179.668,-132.041,168.312,77.428,166.817
C04309=1012.086,179.433,-132.017,168.314,77.438,166.822
C04310=1012.087,179.197,-131.991,168.318,77.448,166.828
C04311=1012.087,178.961,-131.967,168.319,77.457,166.831
C04312=1012.088,178.725,-131.942,168.322,77.467,166.837
C04313=1012.088,178.490,-131.917,168.325,77.476,166.843
C04314=1012.088,178.254,-131.892,168.329,77.486,166.849
C04315=1012.090,178.018,-131.868,168.330,77.495,166.853
C04316=1012.089,177.782,-131.843,168.333,77.505,166.859
C04317=1012.090,177.546,-131.818,168.336,77.513,166.863
C04318=1012.090,177.311,-131.793,168.339,77.523,166.869
C04319=1012.091,177.075,-131.768,168.341,77.534,166.874
C04320=1012.091,176.838,-131.744,168.345,77.544,166.880
C04321=1012.091,176.603,-131.719,168.348,77.553,166.886
C04322=1012.092,176.368,-131.694,168.349,77.562,166.890
C04323=1012.092,176.132,-131.670,168.353,77.572,166.896
C04324=1012.093,175.896,-131.645,168.357,77.581,166.902
C04325=1012.093,175.660,-131.620,168.359,77.590,166.906
C04326=1012.094,175.424,-131.595,168.362,77.600,166.912
C04327=1012.094,175.189,-131.571,168.365,77.609,166.917
C04328=1012.095,174.953,-131.546,168.368,77.618,166.923
C04329=1012.095,174.717,-131.521,168.372,77.628,166.929
C04330=1012.096,174.481,-131.497,168.375,77.638,166.935
C04331=1012.096,174.246,-131.472,168.376,77.647,166.939
C04332=1012.097,174.009,-131.447,168.380,77.657,166.945
C04333=1012.097,173.774,-131.423,168.384,77.667,166.951
C04334=1012.098,173.538,-131.397,168.385,77.676,166.955
C04335=1012.098,173.303,-131.374,168.390,77.685,166.961
C04336=1012.098,173.067,-131.349,168.391,77.694,166.966
C04337=1012.099,172.831,-131.324,168.396,77.703,166.972
C04338=1012.099,172.595,-131.299,168.397,77.712,166.976
C04339=1012.100,172.360,-131.275,168.401,77.722,166.982
C04340=1012.100,172.124,-131.250,168.405,77.732,166.988
C04341=1012.101,171.889,-131.225,168.408,77.741,166.994
C04342=1012.101,171.652,-131.201,168.409,77.751,166.999
C04343=1012.102,171.417,-131.177,168.415,77.760,167.005
C04344=1012.102,171.181,-131.152,168.418,77.769,167.011
C04345=1012.103,170.946,-131.127,168.421,77.778,167.016
C04346=1012.104,170.710,-131.103,168.422,77.787,167.021
C04347=1012.104,170.474,-131.078,168.427,77.796,167.027
C04348=1012.105,170.239,-131.054,168.431,77.806,167.033
C04349=1012.105,170.003,-131.029,168.432,77.815,167.038
C04350=1012.106,169.767,-131.005,168.436,77.825,167.044
C04351=1012.106,169.531,-130.980,168.440,77.835,167.050
C04352=1012.107,169.296,-130.956,168.443,77.843,167.055
C04353=1012.107,169.061,-130.931,168.447,77.853,167.061
C04354=1012.108,168.824,-130.907,168.449,77.861,167.066
C04355=1012.108,168.589,-130.882,168.453,77.871,167.072
C04356=1012.108,168.354,-130.857,168.456,77.879,167.077
C04357=1012.109,168.118,-130.833,168.461,77.889,167.084
C04358=1012.110,167.883,-130.808,168.463,77.898,167.088
C04359=1012.110,167.646,-130.784,168.466,77.907,167.094
C04360=1012.111,167.411,-130.759,168.470,77.917,167.101
C04361=1012.111,167.176,-130.735,168.473,77.926,167.106
C04362=1012.112,166.940,-130.710,168.477,77.936,167.112
C04363=1012.113,166.704,-130.686,168.482,77.945,167.119
C04364=1012.113,166.469,-130.662,168.484,77.954,167.123
C04365=1012.114,166.233,-130.637,168.487,77.962,167.128
C04366=1012.114,165.998,-130.612,168.492,77.971,167.135
C04367=1012.115,165.762,-130.589,168.495,77.980,167.140
C04368=1012.115,165.526,-130.563,168.499,77.990,167.146
C04369=1012.116,165.291,-130.539,168.502,77.998,167.151
C04370=1012.116,164.987,-130.508,168.506,78.010,167.158
C04371=1012.117,164.670,-130.475,168.512,78.022,167.167
C04372=1012.118,164.395,-130.447,168.516,78.032,167.174
C04373=1012.119,164.061,-130.412,168.521,78.046,167.182
C04374=1012.120,163.840,-130.389,168.524,78.054,167.187
C04375=1012.120,163.603,-130.364,168.529,78.063,167.194
C04376=1012.121,163.339,-130.337,168.533,78.073,167.201
C04377=1012.121,163.046,-130.307,168.537,78.085,167.208
C04378=1012.122,162.737,-130.275,168.543,78.096,167.215
C04379=1012.123,162.447,-130.245,168.545,78.107,167.221
C04380=1012.124,162.139,-130.213,168.552,78.119,167.230
C04381=1012.125,161.835,-130.182,168.557,78.131,167.238
C04382=1012.124,161.543,-130.152,168.560,78.141,167.244
C04383=1012.126,161.266,-130.123,168.565,78.152,167.252
C04384=1012.126,161.003,-130.096,168.569,78.162,167.258
C04385=1012.128,160.754,-130.070,168.574,78.172,167.265
C04386=1012.128,160.513,-130.045,168.578,78.182,167.271
C04387=1012.129,160.279,-130.021,168.581,78.190,167.276
C04388=1012.128,160.047,-129.999,168.606,78.230,167.308
C04389=1012.128,159.814,-129.978,168.663,78.318,167.380
C04390=1012.128,159.580,-129.958,168.721,78.406,167.452
C04391=1012.128,159.344,-129.938,168.780,78.494,167.526
C04392=1012.128,159.108,-129.918,168.842,78.584,167.603
C04393=1012.128,158.873,-129.898,168.904,78.672,167.679
C04394=1012.128,158.637,-129.878,168.968,78.760,167.757
C04395=1012.127,158.401,-129.856,169.033,78.849,167.836
C04396=1012.127,158.165,-129.837,169.100,78.937,167.917
C04397=1012.127,157.928,-129.816,169.167,79.026,167.998
C04398=1012.127,157.690,-129.795,169.235,79.115,168.081
C04399=1012.127,157.452,-129.775,169.305,79.204,168.166
C04400=1012.127,157.212,-129.754,169.377,79.293,168.252
C04401=1012.126,156.973,-129.734,169.450,79.383,168.340
C04402=1012.126,156.734,-129.713,169.526,79.472,168.429
C04403=1012.126,156.494,-129.692,169.603,79.561,168.520
C04404=1012.126,156.255,-129.671,169.682,79.650,168.613
C04405=1012.127,156.015,-129.651,169.764,79.739,168.708
C04406=1012.126,155.776,-129.631,169.844,79.827,168.802
C04407=1012.126,155.537,-129.610,169.928,79.917,168.900
C04408=1012.126,155.296,-129.590,170.012,80.005,168.998
C04409=1012.126,155.057,-129.568,170.101,80.095,169.100
C04410=1012.126,154.815,-129.548,170.188,80.183,169.202
C04411=1012.126,154.575,-129.527,170.282,80.273,169.308
C04412=1012.126,154.334,-129.506,170.374,80.361,169.414
C04413=1012.126,154.093,-129.485,170.468,80.450,169.522
C04414=1012.126,153.852,-129.465,170.565,80.539,169.632
C04415=1012.126,153.611,-129.444,170.668,80.628,169.748
C04416=1012.126,153.370,-129.423,170.769,80.717,169.862
C04417=1012.126,153.128,-129.403,170.873,80.805,169.980
C04418=1012.126,152.886,-129.382,170.979,80.895,170.099
C04419=1012.127,152.644,-129.361,171.085,80.983,170.218
C04420=1012.126,152.400,-129.340,171.197,81.071,170.343
C04421=1012.126,152.151,-129.319,171.316,81.163,170.476
C04422=1012.127,151.897,-129.297,171.436,81.256,170.610
C04423=1012.126,151.634,-129.275,171.566,81.351,170.753
C04424=1012.127,151.363,-129.251,171.703,81.450,170.904
C04425=1012.127,151.084,-129.227,171.848,81.551,171.064
C04426=1012.127,150.797,-129.202,171.999,81.655,171.230
C04427=1012.127,150.505,-129.178,172.157,81.760,171.403
C04428=1012.127,150.208,-129.152,172.326,81.868,171.587
C04429=1012.128,149.909,-129.127,172.500,81.976,171.777
C04430=1012.128,149.608,-129.101,172.679,82.084,171.971
C04431=1012.128,149.309,-129.075,172.861,82.192,172.168
C04432=1012.128,149.013,-129.049,173.051,82.298,172.372
C04433=1012.128,148.721,-129.024,173.239,82.402,172.574
C04434=1012.129,148.436,-129.000,173.429,82.505,172.779
C04435=1012.129,148.158,-128.976,173.621,82.604,172.984
C04436=1012.129,147.888,-128.953,173.811,82.700,173.188
C04437=1012.129,147.626,-128.931,174.002,82.793,173.392
C04438=1012.130,147.372,-128.909,174.195,82.884,173.597
C04439=1012.130,147.123,-128.887,174.381,82.971,173.795
C04440=1012.129,146.880,-128.867,174.575,83.057,174.000
C04441=1012.130,146.637,-128.846,174.769,83.143,174.206
C04442=1012.131,146.395,-128.825,174.969,83.228,174.418
C04443=1012.131,146.153,-128.804,175.175,83.313,174.635
C04444=1012.131,145.911,-128.783,175.388,83.398,174.859
C04445=1012.131,145.668,-128.764,175.606,83.483,175.088
C04446=1012.132,145.427,-128.743,175.832,83.567,175.325
C04447=1012.132,145.179,-128.722,176.062,83.653,175.567
C04448=1012.133,144.943,-128.702,176.291,83.735,175.806
C04449=1012.132,144.702,-128.680,176.538,83.819,176.063
C04450=1012.132,144.461,-128.660,176.785,83.903,176.322
C04451=1012.133,144.219,-128.639,177.040,83.987,176.588
C04452=1012.134,143.979,-128.618,177.304,84.070,176.862
C04453=1012.134,143.738,-128.598,177.569,84.152,177.139
C04454=1012.134,143.497,-128.577,177.850,84.234,177.430
C04455=1012.135,143.257,-128.557,178.133,84.317,177.723
C04456=1012.135,143.017,-128.536,178.432,84.399,178.032
C04457=1012.135,142.778,-128.516,178.734,84.480,178.345
C04458=1012.135,142.538,-128.496,179.046,84.561,178.667
C04459=1012.136,142.298,-128.475,179.368,84.642,178.999
C04460=1012.136,142.060,-128.455,179.693,84.723,179.335
C04461=1012.137,141.820,-128.435,-179.964,84.804,179.688
C04462=1012.137,141.575,-128.414,-179.601,84.885,-179.939
C04463=1012.138,141.364,-128.396,-179.284,84.956,-179.613
C04464=1012.138,141.109,-128.373,-178.883,85.041,-179.201
C04465=1012.138,140.937,-128.359,-178.605,85.098,-178.916
C04466=1012.138,140.564,-128.327,-177.979,85.222,-178.275
C04467=1012.140,140.288,-128.303,-177.503,85.311,-177.788
C04468=1012.140,139.993,-128.279,-176.965,85.408,-177.238
C04469=1012.141,139.684,-128.252,-176.374,85.508,-176.635
C04470=1012.141,139.372,-128.225,-175.754,85.609,-176.002
C04471=1012.142,139.064,-128.200,-175.104,85.708,-175.341
C04472=1012.143,138.770,-128.175,-174.464,85.802,-174.689
C04473=1012.143,138.496,-128.151,-173.848,85.888,-174.062
C04474=1012.144,138.244,-128.130,-173.251,85.967,-173.456
C04475=1012.145,137.822,-128.094,-172.192,86.099,-172.380
C04476=1012.146,137.440,-128.061,-171.173,86.217,-171.347
C04477=1012.146,137.023,-128.026,-169.989,86.343,-170.148
C04478=1012.147,136.640,-127.993,-168.822,86.458,-168.966
C04479=1012.148,136.253,-127.960,-167.574,86.571,-167.704
C04480=1012.149,135.834,-127.924,-166.117,86.693,-166.232
C04481=1012.150,135.609,-127.906,-165.299,86.757,-165.406
C04482=1012.150,135.376,-127.886,-164.411,86.822,-164.510
C04483=1012.151,135.091,-127.861,-163.268,86.901,-163.357
C04484=1012.152,134.795,-127.836,-162.023,86.981,-162.103
C04485=1012.152,134.555,-127.816,-160.969,87.046,-161.039
C04486=1012.153,134.320,-127.796,-159.887,87.108,-159.949
C04487=1012.154,134.085,-127.776,-158.763,87.168,-158.817
C04488=1012.154,133.850,-127.756,-157.588,87.227,-157.635
C04489=1012.155,133.614,-127.736,-156.356,87.286,-156.394
C04490=1012.155,133.379,-127.716,-155.075,87.343,-155.106
C04491=1012.156,133.144,-127.696,-153.757,87.398,-153.780
C04492=1012.157,132.909,-127.676,-152.362,87.451,-152.377
C04493=1012.157,132.673,-127.656,-150.906,87.503,-150.913
C04494=1012.158,132.438,-127.636,-149.408,87.554,-149.408
C04495=1012.159,132.202,-127.616,-147.826,87.602,-147.818
C04496=1012.159,131.968,-127.596,-146.200,87.649,-146.185
C04497=1012.160,131.732,-127.576,-144.509,87.694,-144.486
C04498=1012.160,131.497,-127.556,-142.728,87.736,-142.697
C04499=1012.161,131.262,-127.536,-140.902,87.777,-140.864
C04500=1012.162,131.027,-127.516,-139.010,87.814,-138.965
C04501=1012.162,130.791,-127.496,-137.065,87.849,-137.013
C04502=1012.163,130.557,-127.476,-135.044,87.882,-134.984
C04503=1012.164,130.321,-127.456,-132.960,87.912,-132.893
C04504=1012.164,130.086,-127.436,-130.858,87.939,-130.783
C04505=1012.165,129.851,-127.416,-128.660,87.963,-128.579
C04506=1012.166,129.615,-127.397,-126.428,87.984,-126.341
C04507=1012.167,129.322,-127.371,-123.584,88.006,-123.487
C04508=1012.168,128.910,-127.336,-119.529,88.027,-119.420
C04509=1012.169,128.675,-127.317,-117.186,88.035,-117.070
C04510=1012.169,128.439,-127.296,-114.802,88.039,-114.681
C04511=1012.171,128.204,-127.277,-112.416,88.041,-112.287
C04512=1012.171,127.969,-127.257,-110.050,88.039,-109.914
C04513=1012.172,127.734,-127.237,-107.693,88.033,-107.550
C04514=1012.172,127.499,-127.216,-105.352,88.024,-105.203
C04515=1012.173,127.264,-127.197,-103.056,88.011,-102.902
C04516=1012.174,127.028,-127.178,-100.793,87.996,-100.631
C04517=1012.175,126.793,-127.157,-98.545,87.978,-98.377
C04518=1012.175,126.558,-127.138,-96.342,87.956,-96.167
C04519=1012.176,126.323,-127.117,-94.206,87.932,-94.025
C04520=1012.178,126.087,-127.097,-92.125,87.904,-91.938
C04521=1012.178,125.853,-127.078,-90.097,87.874,-89.903
C04522=1012.179,125.618,-127.058,-88.131,87.841,-87.932
C04523=1012.179,125.382,-127.037,-86.222,87.806,-86.016
C04524=1012.180,125.147,-127.018,-84.394,87.769,-84.182
C04525=1012.181,124.912,-126.998,-82.627,87.729,-82.410
C04526=1012.182,124.677,-126.978,-80.904,87.688,-80.681
C04527=1012.183,124.442,-126.959,-79.262,87.644,-79.033
C04528=1012.183,124.206,-126.938,-77.680,87.598,-77.446
C04529=1012.184,123.971,-126.918,-76.159,87.551,-75.919
C04530=1012.185,123.736,-126.898,-74.697,87.502,-74.451
C04531=1012.186,123.501,-126.879,-73.292,87.451,-73.041
C04532=1012.187,123.266,-126.859,-71.951,87.399,-71.694
C04533=1012.188,123.031,-126.839,-70.655,87.346,-70.393
C04534=1012.189,122.796,-126.819,-69.419,87.291,-69.150
C04535=1012.189,122.560,-126.799,-68.225,87.235,-67.951
C04536=1012.190,122.325,-126.779,-67.085,87.178,-66.806
C04537=1012.191,122.090,-126.759,-66.005,87.121,-65.720
C04538=1012.192,121.855,-126.739,-64.949,87.061,-64.659
C04539=1012.193,121.620,-126.720,-63.953,87.002,-63.659
C04540=1012.194,121.385,-126.699,-62.984,86.941,-62.684
C04541=1012.195,121.150,-126.680,-62.066,86.880,-61.761
C04542=1012.196,120.915,-126.660,-61.171,86.817,-60.861
C04543=1012.197,120.680,-126.640,-60.285,86.752,-59.969
///RCONF 0,0,0,0,1,0,0,0,0,0,0,0,0,0,0,0,0,0,0,0,0,0,0,0
C04544=1012.198,120.445,-126.621,-59.402,86.683,-59.082
C04545=1012.199,120.209,-126.601,-58.546,86.612,-58.219
C04546=1012.199,119.974,-126.582,-57.737,86.542,-57.406
C04547=1012.201,119.739,-126.562,-56.949,86.470,-56.612
C04548=1012.201,119.504,-126.543,-56.203,86.398,-55.861
C04549=1012.202,119.269,-126.523,-55.478,86.326,-55.131
C04550=1012.204,119.033,-126.503,-54.792,86.253,-54.440
C04551=1012.204,118.798,-126.484,-54.132,86.180,-53.774
C04552=1012.205,118.563,-126.464,-53.495,86.105,-53.134
C04553=1012.206,118.328,-126.445,-52.885,86.031,-52.519
C04554=1012.207,118.093,-126.425,-52.289,85.956,-51.917
C04555=1012.208,117.857,-126.406,-51.723,85.880,-51.346
C04556=1012.209,117.623,-126.386,-51.177,85.805,-50.796
C04557=1012.210,117.387,-126.366,-50.652,85.730,-50.266
C04558=1012.211,117.152,-126.347,-50.153,85.654,-49.763
C04559=1012.212,116.917,-126.327,-49.664,85.577,-49.269
C04560=1012.212,116.682,-126.308,-49.191,85.500,-48.792
C04561=1012.214,116.446,-126.289,-48.736,85.423,-48.331
C04562=1012.214,116.211,-126.269,-48.302,85.346,-47.894
C04563=1012.216,115.977,-126.250,-47.876,85.269,-47.463
C04564=1012.217,115.741,-126.230,-47.470,85.192,-47.053
C04565=1012.218,115.506,-126.211,-47.072,85.114,-46.650
C04566=1012.219,115.271,-126.191,-46.692,85.035,-46.267
C04567=1012.219,115.036,-126.172,-46.324,84.957,-45.896
C04568=1012.221,114.801,-126.152,-45.968,84.879,-45.535
C04569=1012.222,114.565,-126.132,-45.617,84.801,-45.180
C04570=1012.223,114.330,-126.113,-45.282,84.723,-44.840
C04571=1012.224,114.095,-126.093,-44.957,84.644,-44.512
C04572=1012.225,113.860,-126.074,-44.648,84.566,-44.200
C04573=1012.226,113.625,-126.055,-44.342,84.488,-43.889
C04574=1012.228,113.390,-126.035,-44.045,84.409,-43.589
C04575=1012.229,113.022,-126.005,-43.600,84.285,-43.138
C04576=1012.231,112.684,-125.977,-43.208,84.172,-42.741
C04577=1012.231,112.449,-125.958,-42.947,84.093,-42.477
C04578=1012.232,112.214,-125.937,-42.689,84.014,-42.215
C04579=1012.234,111.979,-125.918,-42.442,83.935,-41.965
C04580=1012.235,111.744,-125.899,-42.202,83.856,-41.722
C04581=1012.236,111.509,-125.879,-41.968,83.777,-41.485
C04582=1012.237,111.274,-125.859,-41.741,83.698,-41.254
C04583=1012.238,111.039,-125.840,-41.519,83.619,-41.029
C04584=1012.239,110.803,-125.820,-41.302,83.540,-40.809
C04585=1012.240,110.568,-125.801,-41.091,83.460,-40.595
C04586=1012.242,110.333,-125.782,-40.886,83.381,-40.387
C04587=1012.243,110.098,-125.762,-40.685,83.302,-40.183
C04588=1012.243,109.863,-125.743,-40.492,83.223,-39.988
C04589=1012.245,109.627,-125.723,-40.301,83.143,-39.794
C04590=1012.246,109.392,-125.704,-40.118,83.064,-39.609
C04591=1012.247,109.157,-125.684,-39.936,82.985,-39.423
C04592=1012.248,108.922,-125.665,-39.761,82.906,-39.246
C04593=1012.250,108.687,-125.646,-39.590,82.827,-39.072
C04594=1012.251,108.452,-125.626,-39.423,82.748,-38.903
C04595=1012.251,108.216,-125.607,-39.260,82.669,-38.738
C04596=1012.253,107.981,-125.587,-39.100,82.590,-38.575
C04597=1012.254,107.746,-125.567,-38.944,82.511,-38.417
C04598=1012.255,107.511,-125.549,-38.791,82.433,-38.261
C04599=1012.256,107.276,-125.529,-38.642,82.353,-38.110
C04600=1012.258,107.041,-125.509,-38.498,82.275,-37.964
C04601=1012.258,106.805,-125.490,-38.356,82.195,-37.819
C04602=1012.260,106.570,-125.470,-38.218,82.117,-37.680
C04603=1012.261,106.336,-125.450,-38.080,82.038,-37.540
C04604=1012.262,106.101,-125.431,-37.948,81.960,-37.406
C04605=1012.263,105.865,-125.411,-37.819,81.881,-37.275
C04606=1012.264,105.630,-125.392,-37.690,81.802,-37.143
C04607=1012.266,105.395,-125.372,-37.566,81.723,-37.018
C04608=1012.267,105.160,-125.353,-37.445,81.645,-36.895
C04609=1012.268,104.925,-125.334,-37.326,81.566,-36.774
C04610=1012.269,104.690,-125.314,-37.211,81.489,-36.657
C04611=1012.271,104.454,-125.294,-37.096,81.410,-36.542
C04612=1012.271,104.219,-125.275,-36.983,81.332,-36.426
C04613=1012.273,103.984,-125.256,-36.876,81.254,-36.318
C04614=1012.274,103.749,-125.236,-36.767,81.175,-36.207
C04615=1012.276,103.513,-125.217,-36.663,81.097,-36.103
C04616=1012.276,103.278,-125.198,-36.558,81.019,-35.997
C04617=1012.278,103.043,-125.178,-36.458,80.941,-35.895
C04618=1012.280,102.808,-125.159,-36.359,80.863,-35.795
C04619=1012.281,102.572,-125.139,-36.262,80.786,-35.697
C04620=1012.282,102.337,-125.119,-36.167,80.708,-35.601
C04621=1012.283,102.102,-125.100,-36.074,80.630,-35.507
C04622=1012.284,101.867,-125.081,-35.981,80.553,-35.412
C04623=1012.286,101.632,-125.061,-35.891,80.475,-35.321
C04624=1012.287,101.396,-125.041,-35.805,80.398,-35.235
C04625=1012.288,101.161,-125.022,-35.717,80.320,-35.145
C04626=1012.289,100.926,-125.003,-35.633,80.244,-35.060
C04627=1012.290,100.691,-124.983,-35.549,80.166,-34.975
C04628=1012.292,100.456,-124.964,-35.467,80.089,-34.893
C04629=1012.293,100.221,-124.944,-35.387,80.012,-34.812
C04630=1012.294,99.985,-124.925,-35.308,79.936,-34.733
C04631=1012.295,99.750,-124.905,-35.232,79.858,-34.657
C04632=1012.297,99.515,-124.886,-35.156,79.781,-34.580
C04633=1012.298,99.280,-124.866,-35.080,79.705,-34.503
C04634=1012.300,99.045,-124.846,-35.006,79.628,-34.429
C04635=1012.300,98.810,-124.827,-34.934,79.551,-34.356
C04636=1012.302,98.574,-124.807,-34.864,79.475,-34.287
C04637=1012.303,98.339,-124.788,-34.793,79.399,-34.215
C04638=1012.305,98.104,-124.768,-34.726,79.322,-34.148
C04639=1012.306,97.869,-124.749,-34.657,79.246,-34.078
C04640=1012.308,97.633,-124.730,-34.592,79.170,-34.014
C04641=1012.308,97.398,-124.711,-34.527,79.094,-33.948
C04642=1012.310,97.163,-124.691,-34.463,79.018,-33.884
C04643=1012.311,96.927,-124.672,-34.400,78.943,-33.821
C04644=1012.313,96.692,-124.652,-34.338,78.867,-33.759
C04645=1012.314,96.457,-124.632,-34.277,78.791,-33.697
C04646=1012.316,96.137,-124.606,-34.197,78.688,-33.618
C04647=1012.318,95.752,-124.574,-34.102,78.565,-33.524
C04648=1012.319,95.516,-124.554,-34.044,78.489,-33.467
C04649=1012.320,95.281,-124.535,-33.988,78.415,-33.411
C04650=1012.322,95.045,-124.515,-33.934,78.340,-33.357
C04651=1012.323,94.809,-124.496,-33.880,78.265,-33.303
C04652=1012.325,94.575,-124.476,-33.827,78.190,-33.251
C04653=1012.326,94.339,-124.457,-33.774,78.115,-33.198
C04654=1012.328,94.104,-124.437,-33.722,78.041,-33.146
C04655=1012.328,93.869,-124.418,-33.670,77.966,-33.095
C04656=1012.329,93.633,-124.398,-33.620,77.891,-33.047
C04657=1012.331,93.399,-124.379,-33.572,77.817,-32.999
C04658=1012.333,93.163,-124.359,-33.522,77.742,-32.950
C04659=1012.334,92.928,-124.339,-33.474,77.669,-32.902
C04660=1012.335,92.692,-124.320,-33.428,77.595,-32.857
C04661=1012.337,92.456,-124.301,-33.382,77.521,-32.812
C04662=1012.338,92.221,-124.281,-33.336,77.447,-32.768
C04663=1012.340,91.986,-124.262,-33.291,77.374,-32.723
C04664=1012.341,91.751,-124.242,-33.247,77.300,-32.681
C04665=1012.342,91.516,-124.223,-33.202,77.227,-32.637
C04666=1012.343,91.281,-124.203,-33.158,77.153,-32.593
C04667=1012.344,91.045,-124.183,-33.117,77.080,-32.555
C04668=1012.346,90.785,-124.162,-33.071,76.999,-32.510
C04669=1012.348,90.467,-124.136,-33.014,76.901,-32.454
C04670=1012.350,90.133,-124.108,-32.957,76.797,-32.399
C04671=1012.352,89.849,-124.085,-32.910,76.710,-32.354
C04672=1012.354,89.612,-124.065,-32.870,76.636,-32.315
C04673=1012.355,89.379,-124.045,-32.832,76.565,-32.278
C04674=1012.356,89.149,-124.027,-32.796,76.495,-32.244
C04675=1012.357,88.923,-124.008,-32.760,76.425,-32.209
C04676=1012.359,88.698,-123.989,-32.725,76.356,-32.176
C04677=1012.360,88.474,-123.970,-32.690,76.288,-32.142
C04678=1012.361,88.250,-123.951,-32.656,76.219,-32.110
C04679=1012.363,88.026,-123.933,-32.622,76.150,-32.078
C04680=1012.364,87.798,-123.914,-32.588,76.082,-32.045
C04681=1012.365,87.568,-123.895,-32.555,76.011,-32.014
C04682=1012.366,87.334,-123.876,-32.521,75.940,-31.982
C04683=1012.368,87.098,-123.857,-32.487,75.869,-31.950
C04684=1012.369,86.860,-123.836,-32.454,75.797,-31.919
C04685=1012.371,86.622,-123.816,-32.420,75.725,-31.886
C04686=1012.372,86.382,-123.797,-32.388,75.653,-31.857
C04687=1012.373,86.143,-123.777,-32.356,75.581,-31.827
C04688=1012.375,85.903,-123.757,-32.323,75.509,-31.796
C04689=1012.377,85.663,-123.737,-32.292,75.437,-31.766
C04690=1012.378,85.422,-123.717,-32.262,75.365,-31.739
C04691=1012.379,85.181,-123.697,-32.230,75.293,-31.709
C04692=1012.380,84.939,-123.677,-32.200,75.221,-31.681
C04693=1012.382,84.697,-123.656,-32.170,75.150,-31.654
C04694=1012.383,84.455,-123.636,-32.140,75.076,-31.626
C04695=1012.385,84.212,-123.617,-32.111,75.005,-31.600
C04696=1012.387,83.968,-123.597,-32.082,74.933,-31.573
C04697=1012.388,83.723,-123.576,-32.052,74.860,-31.545
C04698=1012.390,83.479,-123.555,-32.024,74.789,-31.520
C04699=1012.391,83.234,-123.536,-31.996,74.717,-31.494
C04700=1012.393,82.989,-123.515,-31.969,74.644,-31.471
C04701=1012.394,82.743,-123.494,-31.941,74.573,-31.446
C04702=1012.396,82.497,-123.474,-31.914,74.501,-31.422
C04703=1012.397,82.251,-123.453,-31.886,74.428,-31.396
C04704=1012.399,82.005,-123.433,-31.860,74.356,-31.373
C04705=1012.400,81.758,-123.412,-31.834,74.284,-31.349
C04706=1012.401,81.511,-123.392,-31.808,74.214,-31.326
C04707=1012.403,81.267,-123.372,-31.783,74.143,-31.305
C04708=1012.404,81.039,-123.353,-31.760,74.077,-31.284
C04709=1012.406,80.822,-123.335,-31.738,74.014,-31.265
C04710=1012.407,80.605,-123.317,-31.716,73.952,-31.246
C04711=1012.409,80.376,-123.298,-31.693,73.886,-31.226
C04712=1012.410,80.133,-123.277,-31.669,73.817,-31.204
C04713=1012.411,79.886,-123.257,-31.646,73.746,-31.185
C04714=1012.412,79.642,-123.237,-31.622,73.677,-31.164
C04715=1012.415,79.400,-123.216,-31.600,73.607,-31.145
C04716=1012.416,79.160,-123.197,-31.578,73.539,-31.127
C04717=1012.417,78.922,-123.177,-31.555,73.472,-31.106
C04718=1012.418,78.688,-123.157,-31.534,73.405,-31.088
C04719=1012.420,78.455,-123.138,-31.513,73.340,-31.071
C04720=1012.421,78.225,-123.118,-31.492,73.275,-31.053
C04721=1012.422,77.997,-123.100,-31.473,73.210,-31.037
C04722=1012.423,77.769,-123.081,-31.453,73.146,-31.021
C04723=1012.426,77.433,-123.053,-31.424,73.052,-30.997
C04724=1012.428,77.085,-123.024,-31.395,72.955,-30.973
C04725=1012.429,76.855,-123.005,-31.376,72.890,-30.957
C04726=1012.431,76.622,-122.986,-31.357,72.826,-30.942
C04727=1012.432,76.387,-122.966,-31.338,72.761,-30.926
C04728=1012.434,76.149,-122.945,-31.319,72.695,-30.912
C04729=1012.435,75.907,-122.926,-31.300,72.628,-30.896
C04730=1012.437,75.664,-122.906,-31.281,72.562,-30.881
C04731=1012.439,75.418,-122.885,-31.262,72.493,-30.865
C04732=1012.440,75.171,-122.865,-31.242,72.426,-30.849
C04733=1012.441,74.922,-122.844,-31.225,72.358,-30.836
C04734=1012.443,74.663,-122.822,-31.205,72.288,-30.820
C04735=1012.445,74.391,-122.799,-31.185,72.213,-30.805
C04736=1012.445,74.124,-122.777,-31.166,72.141,-30.790
C04737=1012.447,73.873,-122.756,-31.148,72.073,-30.777
C04738=1012.449,73.626,-122.736,-31.130,72.007,-30.761
C04739=1012.450,73.380,-122.716,-31.113,71.941,-30.749
C04740=1012.452,73.135,-122.694,-31.096,71.875,-30.737
C04741=1012.453,72.891,-122.674,-31.079,71.809,-30.724
C04742=1012.455,72.648,-122.654,-31.063,71.745,-30.712
C04743=1012.457,72.405,-122.634,-31.046,71.680,-30.699
C04744=1012.458,72.163,-122.615,-31.030,71.615,-30.688
C04745=1012.459,71.921,-122.593,-31.015,71.552,-30.676
C04746=1012.461,71.679,-122.574,-30.999,71.488,-30.665
C04747=1012.461,71.438,-122.553,-30.984,71.425,-30.654
C04748=1012.463,71.197,-122.534,-30.968,71.361,-30.641
C04749=1012.465,70.955,-122.513,-30.953,71.297,-30.632
C04750=1012.466,70.715,-122.493,-30.938,71.234,-30.621
C04751=1012.468,70.473,-122.473,-30.924,71.172,-30.612
C04752=1012.469,70.233,-122.453,-30.910,71.109,-30.602
C04753=1012.471,69.992,-122.433,-30.894,71.047,-30.590
C04754=1012.472,69.750,-122.413,-30.881,70.985,-30.581
C04755=1012.473,69.510,-122.393,-30.866,70.922,-30.571
C04756=1012.475,69.267,-122.372,-30.852,70.860,-30.561
C04757=1012.476,69.021,-122.352,-30.838,70.796,-30.553
C04758=1012.478,68.772,-122.331,-30.824,70.733,-30.544
C04759=1012.479,68.523,-122.311,-30.810,70.669,-30.533
C04760=1012.481,68.274,-122.290,-30.796,70.606,-30.524
C04761=1012.483,68.028,-122.270,-30.783,70.544,-30.516
C04762=1012.483,67.787,-122.249,-30.770,70.483,-30.508
C04763=1012.486,67.548,-122.229,-30.757,70.423,-30.500
C04764=1012.486,67.311,-122.209,-30.744,70.363,-30.491
C04765=1012.488,67.073,-122.190,-30.732,70.304,-30.483
C04766=1012.489,66.837,-122.169,-30.719,70.244,-30.475
C04767=1012.491,66.601,-122.150,-30.707,70.185,-30.468
C04768=1012.492,66.387,-122.132,-30.697,70.133,-30.462
C04769=1012.494,65.995,-122.099,-30.676,70.035,-30.449
C04770=1012.496,65.763,-122.080,-30.665,69.979,-30.443
C04771=1012.497,65.520,-122.059,-30.653,69.918,-30.436
C04772=1012.499,65.266,-122.039,-30.641,69.856,-30.428
C04773=1012.501,65.006,-122.017,-30.629,69.792,-30.422
C04774=1012.502,64.741,-121.995,-30.616,69.727,-30.415
C04775=1012.504,64.470,-121.972,-30.603,69.662,-30.407
C04776=1012.504,64.203,-121.950,-30.590,69.597,-30.400
C04777=1012.507,63.951,-121.929,-30.579,69.536,-30.394
C04778=1012.508,63.712,-121.909,-30.569,69.479,-30.389
C04779=1012.510,63.462,-121.887,-30.557,69.419,-30.382
C04780=1012.511,63.179,-121.865,-30.544,69.351,-30.376
C04781=1012.512,62.883,-121.840,-30.531,69.281,-30.368
C04782=1012.514,62.608,-121.817,-30.519,69.216,-30.362
C04783=1012.516,62.320,-121.792,-30.506,69.147,-30.356
C04784=1012.518,62.044,-121.769,-30.495,69.082,-30.350
C04785=1012.519,61.809,-121.750,-30.485,69.027,-30.345
C04786=1012.520,61.573,-121.730,-30.475,68.971,-30.340
C04787=1012.521,61.336,-121.711,-30.465,68.916,-30.336
C04788=1012.523,61.101,-121.691,-30.456,68.862,-30.332
C04789=1012.525,60.865,-121.671,-30.446,68.807,-30.326
C04790=1012.526,60.630,-121.651,-30.437,68.753,-30.323
C04791=1012.527,60.394,-121.632,-30.428,68.698,-30.320
C04792=1012.528,60.158,-121.612,-30.418,68.644,-30.314
C04793=1012.529,59.922,-121.592,-30.409,68.589,-30.311
C04794=1012.531,59.687,-121.572,-30.400,68.536,-30.307
C04795=1012.533,59.451,-121.552,-30.391,68.482,-30.303
C04796=1012.534,59.215,-121.533,-30.382,68.429,-30.299
C04797=1012.535,58.979,-121.513,-30.373,68.376,-30.296
C04798=1012.536,58.744,-121.493,-30.364,68.322,-30.291
C04799=1012.538,58.508,-121.474,-30.356,68.269,-30.288
C04800=1012.539,58.273,-121.454,-30.347,68.216,-30.286
C04801=1012.540,58.037,-121.435,-30.338,68.164,-30.281
C04802=1012.542,57.801,-121.414,-30.330,68.111,-30.279
C04803=1012.543,57.565,-121.394,-30.322,68.060,-30.276
C04804=1012.544,57.330,-121.375,-30.313,68.007,-30.273
C04805=1012.546,57.094,-121.355,-30.305,67.955,-30.270
C04806=1012.547,56.858,-121.336,-30.298,67.903,-30.269
C04807=1012.548,56.622,-121.316,-30.289,67.851,-30.265
C04808=1012.549,56.387,-121.296,-30.281,67.800,-30.262
C04809=1012.551,56.151,-121.276,-30.274,67.749,-30.261
C04810=1012.553,55.916,-121.256,-30.266,67.698,-30.258
C04811=1012.554,55.680,-121.236,-30.257,67.647,-30.254
C04812=1012.555,55.444,-121.217,-30.250,67.596,-30.253
C04813=1012.556,55.208,-121.197,-30.242,67.545,-30.251
C04814=1012.557,54.973,-121.178,-30.234,67.495,-30.248
C04815=1012.559,54.737,-121.158,-30.227,67.445,-30.247
C04816=1012.560,54.502,-121.138,-30.220,67.395,-30.244
C04817=1012.562,54.091,-121.104,-30.207,67.308,-30.242
C04818=1012.564,53.794,-121.079,-30.197,67.246,-30.238
C04819=1012.566,53.559,-121.059,-30.191,67.196,-30.238
C04820=1012.566,53.323,-121.039,-30.184,67.148,-30.236
C04821=1012.568,53.087,-121.019,-30.177,67.099,-30.235
C04822=1012.569,52.852,-121.000,-30.170,67.050,-30.234
C04823=1012.570,52.616,-120.980,-30.163,67.001,-30.233
C04824=1012.572,52.380,-120.961,-30.156,66.953,-30.230
C04825=1012.572,52.144,-120.941,-30.150,66.905,-30.231
C04826=1012.574,51.909,-120.921,-30.142,66.856,-30.228
C04827=1012.576,51.673,-120.901,-30.136,66.809,-30.227
C04828=1012.577,51.438,-120.881,-30.129,66.762,-30.226
C04829=1012.578,51.202,-120.861,-30.123,66.713,-30.226
C04830=1012.579,50.966,-120.841,-30.117,66.666,-30.225
C04831=1012.580,50.731,-120.822,-30.110,66.618,-30.224
C04832=1012.582,50.496,-120.802,-30.104,66.573,-30.223
C04833=1012.583,50.260,-120.783,-30.097,66.525,-30.222
C04834=1012.584,50.024,-120.763,-30.091,66.479,-30.222
C04835=1012.585,49.788,-120.743,-30.084,66.432,-30.220
C04836=1012.586,49.553,-120.723,-30.078,66.385,-30.220
C04837=1012.588,49.317,-120.704,-30.072,66.339,-30.219
C04838=1012.589,49.082,-120.684,-30.066,66.294,-30.219
C04839=1012.590,48.846,-120.664,-30.061,66.248,-30.220
C04840=1012.592,48.611,-120.645,-30.055,66.203,-30.220
C04841=1012.592,48.375,-120.625,-30.049,66.157,-30.219
C04842=1012.594,48.140,-120.605,-30.043,66.112,-30.219
C04843=1012.595,47.904,-120.585,-30.037,66.067,-30.219
C04844=1012.597,47.668,-120.565,-30.031,66.022,-30.218
C04845=1012.598,47.433,-120.545,-30.026,65.977,-30.218
C04846=1012.599,47.197,-120.525,-30.021,65.933,-30.220
C04847=1012.600,46.962,-120.505,-30.015,65.889,-30.219
C04848=1012.601,46.726,-120.486,-30.009,65.845,-30.219
C04849=1012.603,46.491,-120.466,-30.003,65.800,-30.219
C04850=1012.604,46.255,-120.446,-29.998,65.757,-30.219
C04851=1012.605,46.020,-120.426,-29.993,65.713,-30.219
C04852=1012.606,45.784,-120.406,-29.987,65.670,-30.220
C04853=1012.607,45.548,-120.387,-29.982,65.627,-30.221
C04854=1012.609,45.313,-120.367,-29.977,65.584,-30.221
C04855=1012.610,45.078,-120.347,-29.972,65.541,-30.222
C04856=1012.611,44.842,-120.328,-29.966,65.499,-30.221
C04857=1012.612,44.607,-120.308,-29.961,65.456,-30.223
C04858=1012.613,44.371,-120.288,-29.956,65.414,-30.222
C04859=1012.614,44.135,-120.268,-29.951,65.371,-30.224
C04860=1012.616,43.900,-120.248,-29.947,65.330,-30.225
C04861=1012.616,43.665,-120.229,-29.941,65.288,-30.225
C04862=1012.617,43.430,-120.209,-29.937,65.247,-30.226
C04863=1012.619,43.194,-120.190,-29.932,65.205,-30.228
C04864=1012.619,42.958,-120.170,-29.927,65.165,-30.227
C04865=1012.621,42.723,-120.150,-29.922,65.123,-30.228
C04866=1012.622,42.487,-120.130,-29.917,65.082,-30.230
C04867=1012.623,42.252,-120.111,-29.913,65.041,-30.231
C04868=1012.625,42.016,-120.091,-29.908,65.002,-30.232
C04869=1012.626,41.781,-120.071,-29.904,64.961,-30.233
C04870=1012.627,41.546,-120.051,-29.899,64.921,-30.234
C04871=1012.628,41.310,-120.031,-29.895,64.881,-30.236
C04872=1012.629,41.074,-120.012,-29.890,64.842,-30.237
C04873=1012.630,40.839,-119.991,-29.886,64.802,-30.238
C04874=1012.631,40.604,-119.971,-29.881,64.763,-30.239
C04875=1012.633,40.369,-119.952,-29.877,64.723,-30.240
C04876=1012.634,40.133,-119.932,-29.873,64.685,-30.242
C04877=1012.635,39.898,-119.913,-29.869,64.647,-30.243
C04878=1012.635,39.662,-119.893,-29.864,64.607,-30.244
C04879=1012.637,39.427,-119.873,-29.860,64.569,-30.246
C04880=1012.638,39.191,-119.853,-29.856,64.531,-30.247
C04881=1012.639,38.956,-119.834,-29.852,64.494,-30.249
C04882=1012.640,38.721,-119.813,-29.848,64.455,-30.251
C04883=1012.641,38.486,-119.794,-29.843,64.417,-30.252
C04884=1012.643,38.250,-119.774,-29.840,64.380,-30.254
C04885=1012.643,38.014,-119.754,-29.836,64.343,-30.255
C04886=1012.644,37.779,-119.735,-29.832,64.306,-30.257
C04887=1012.645,37.544,-119.715,-29.828,64.269,-30.259
C04888=1012.646,37.308,-119.695,-29.824,64.232,-30.261
C04889=1012.648,37.073,-119.676,-29.820,64.196,-30.261
C04890=1012.649,36.838,-119.655,-29.817,64.160,-30.264
C04891=1012.650,36.603,-119.635,-29.812,64.124,-30.265
C04892=1012.651,36.367,-119.615,-29.809,64.087,-30.268
C04893=1012.651,36.132,-119.596,-29.805,64.052,-30.269
C04894=1012.653,35.896,-119.577,-29.801,64.017,-30.271
C04895=1012.654,35.661,-119.557,-29.798,63.981,-30.273
C04896=1012.655,35.426,-119.536,-29.794,63.947,-30.275
C04897=1012.656,35.191,-119.517,-29.791,63.911,-30.277
C04898=1012.657,34.955,-119.497,-29.787,63.877,-30.279
C04899=1012.658,34.720,-119.478,-29.784,63.841,-30.281
C04900=1012.659,34.484,-119.458,-29.780,63.808,-30.282
C04901=1012.660,34.249,-119.437,-29.777,63.773,-30.285
C04902=1012.661,34.014,-119.418,-29.774,63.740,-30.287
C04903=1012.662,33.778,-119.398,-29.770,63.705,-30.290
C04904=1012.663,33.543,-119.379,-29.767,63.672,-30.291
C04905=1012.664,33.308,-119.359,-29.763,63.639,-30.294
C04906=1012.665,33.073,-119.339,-29.760,63.606,-30.296
C04907=1012.666,32.837,-119.319,-29.757,63.572,-30.297
C04908=1012.667,32.602,-119.299,-29.754,63.540,-30.300
C04909=1012.667,32.367,-119.280,-29.751,63.507,-30.303
C04910=1012.668,32.132,-119.259,-29.747,63.475,-30.304
C04911=1012.670,31.896,-119.240,-29.744,63.442,-30.306
C04912=1012.671,31.661,-119.220,-29.741,63.410,-30.308
C04913=1012.672,31.426,-119.201,-29.738,63.378,-30.311
C04914=1012.672,31.190,-119.181,-29.735,63.347,-30.313
C04915=1012.673,30.955,-119.160,-29.732,63.315,-30.315
C04916=1012.675,30.720,-119.141,-29.729,63.283,-30.319
C04917=1012.675,30.485,-119.121,-29.726,63.252,-30.321
C04918=1012.676,30.249,-119.102,-29.723,63.222,-30.322
C04919=1012.677,30.014,-119.081,-29.720,63.191,-30.324
C04920=1012.679,29.779,-119.062,-29.718,63.160,-30.327
C04921=1012.679,29.543,-119.042,-29.715,63.130,-30.330
C04922=1012.680,29.308,-119.022,-29.712,63.100,-30.332
C04923=1012.681,29.073,-119.002,-29.709,63.070,-30.335
C04924=1012.682,28.838,-118.982,-29.706,63.040,-30.337
C04925=1012.683,28.603,-118.963,-29.704,63.011,-30.339
C04926=1012.684,28.368,-118.943,-29.701,62.981,-30.343
C04927=1012.684,28.134,-118.923,-29.698,62.952,-30.345
C04928=1012.685,27.900,-118.904,-29.695,62.924,-30.346
C04929=1012.686,27.667,-118.884,-29.693,62.895,-30.349
C04930=1012.688,27.433,-118.864,-29.691,62.867,-30.352
C04931=1012.688,27.198,-118.844,-29.688,62.838,-30.355
C04932=1012.689,26.964,-118.825,-29.686,62.810,-30.357
C04933=1012.690,26.730,-118.805,-29.683,62.782,-30.360
C04934=1012.690,26.495,-118.785,-29.681,62.754,-30.362
C04935=1012.691,26.258,-118.765,-29.678,62.726,-30.366
C04936=1012.693,26.021,-118.745,-29.676,62.699,-30.368
C04937=1012.693,25.784,-118.726,-29.673,62.672,-30.370
C04938=1012.694,25.547,-118.706,-29.671,62.644,-30.372
C04939=1012.695,25.310,-118.685,-29.668,62.617,-30.374
C04940=1012.696,25.075,-118.666,-29.666,62.591,-30.378
C04941=1012.697,24.840,-118.646,-29.664,62.564,-30.381
C04942=1012.698,24.604,-118.626,-29.662,62.538,-30.384
C04943=1012.698,24.367,-118.606,-29.660,62.512,-30.386
C04944=1012.699,24.137,-118.587,-29.658,62.486,-30.389
C04945=1012.700,23.914,-118.568,-29.655,62.462,-30.390
C04946=1012.700,23.704,-118.551,-29.654,62.439,-30.394
C04947=1012.702,23.341,-118.520,-29.650,62.401,-30.397
C04948=1012.703,23.040,-118.494,-29.648,62.368,-30.401
C04949=1012.703,22.749,-118.470,-29.645,62.338,-30.404
C04950=1012.705,22.404,-118.441,-29.642,62.301,-30.408
C04951=1012.706,21.991,-118.407,-29.638,62.259,-30.413
C04952=1012.708,21.580,-118.371,-29.635,62.218,-30.418
C04953=1012.708,21.321,-118.350,-29.633,62.192,-30.420
C04954=1012.710,21.031,-118.325,-29.631,62.164,-30.424
C04955=1012.710,20.722,-118.300,-29.628,62.134,-30.427
C04956=1012.712,20.403,-118.273,-29.626,62.103,-30.431
C04957=1012.712,20.085,-118.246,-29.623,62.072,-30.434
C04958=1012.713,19.783,-118.220,-29.621,62.044,-30.438
C04959=1012.714,19.388,-118.188,-29.619,62.007,-30.444
C04960=1012.716,19.083,-118.161,-29.617,61.979,-30.448
C04961=1012.716,18.822,-118.139,-29.615,61.956,-30.450
C04962=1012.717,18.588,-118.120,-29.613,61.934,-30.452
C04963=1012.717,18.354,-118.100,-29.611,61.913,-30.455
C04964=1012.719,18.122,-118.080,-29.610,61.893,-30.458
C04965=1012.719,17.890,-118.061,-29.608,61.873,-30.462
C04966=1012.719,17.658,-118.042,-29.607,61.853,-30.463
C04967=1012.720,17.427,-118.022,-29.605,61.833,-30.467
C04968=1012.721,17.196,-118.003,-29.603,61.813,-30.468
C04969=1012.722,16.966,-117.983,-29.602,61.793,-30.472
C04970=1012.722,16.737,-117.964,-29.601,61.774,-30.474
C04971=1012.723,16.509,-117.944,-29.600,61.756,-30.478
C04972=1012.724,16.281,-117.926,-29.598,61.737,-30.480
C04973=1012.725,16.054,-117.906,-29.597,61.719,-30.483
C04974=1012.725,15.826,-117.887,-29.596,61.701,-30.485
C04975=1012.725,15.600,-117.868,-29.595,61.683,-30.488
C04976=1012.726,15.374,-117.849,-29.593,61.666,-30.490
C04977=1012.727,15.147,-117.830,-29.592,61.648,-30.494
C04978=1012.727,14.921,-117.811,-29.591,61.631,-30.496
C04979=1012.728,14.695,-117.792,-29.590,61.614,-30.498
C04980=1012.728,14.469,-117.773,-29.588,61.597,-30.501
C04981=1012.729,14.242,-117.754,-29.587,61.580,-30.504
C04982=1012.730,14.016,-117.735,-29.586,61.564,-30.507
C04983=1012.730,13.789,-117.716,-29.585,61.547,-30.510
C04984=1012.731,13.561,-117.697,-29.584,61.531,-30.512
C04985=1012.731,13.334,-117.677,-29.583,61.515,-30.514
C04986=1012.731,13.106,-117.658,-29.582,61.499,-30.518
C04987=1012.732,12.878,-117.639,-29.581,61.483,-30.519
C04988=1012.733,12.604,-117.616,-29.580,61.464,-30.524
C04989=1012.734,12.192,-117.582,-29.578,61.438,-30.527
C04990=1012.735,11.965,-117.563,-29.577,61.423,-30.530
C04991=1012.735,11.741,-117.544,-29.576,61.408,-30.532
C04992=1012.736,11.523,-117.526,-29.575,61.394,-30.535
C04993=1012.737,11.307,-117.507,-29.574,61.381,-30.537
C04994=1012.737,11.091,-117.489,-29.574,61.366,-30.540
C04995=1012.737,10.873,-117.471,-29.573,61.354,-30.543
C04996=1012.737,10.652,-117.452,-29.572,61.341,-30.545
C04997=1012.738,10.427,-117.433,-29.571,61.327,-30.548
C04998=1012.739,10.202,-117.414,-29.570,61.313,-30.550
C04999=1012.739,9.978,-117.395,-29.570,61.301,-30.553
C05000=1012.739,9.755,-117.376,-29.569,61.288,-30.555
C05001=1012.740,9.532,-117.358,-29.568,61.275,-30.557
C05002=1012.741,9.309,-117.339,-29.568,61.263,-30.560
C05003=1012.742,9.086,-117.320,-29.567,61.251,-30.564
C05004=1012.741,8.864,-117.302,-29.567,61.239,-30.567
C05005=1012.742,8.642,-117.282,-29.566,61.227,-30.568
C05006=1012.743,8.419,-117.264,-29.566,61.215,-30.571
C05007=1012.743,8.196,-117.245,-29.565,61.204,-30.573
C05008=1012.743,7.973,-117.226,-29.564,61.193,-30.575
C05009=1012.744,7.749,-117.207,-29.564,61.181,-30.579
C05010=1012.744,7.523,-117.188,-29.563,61.170,-30.581
C05011=1012.745,7.297,-117.169,-29.563,61.160,-30.583
C05012=1012.745,7.069,-117.150,-29.562,61.149,-30.585
C05013=1012.746,6.840,-117.130,-29.562,61.139,-30.589
C05014=1012.746,6.609,-117.111,-29.561,61.128,-30.591
C05015=1012.747,6.377,-117.092,-29.561,61.118,-30.594
C05016=1012.747,6.143,-117.072,-29.561,61.107,-30.596
C05017=1012.748,5.909,-117.052,-29.560,61.098,-30.598
C05018=1012.748,5.674,-117.033,-29.560,61.088,-30.601
C05019=1012.748,5.442,-117.013,-29.559,61.079,-30.603
C05020=1012.749,5.209,-116.993,-29.559,61.069,-30.606
C05021=1012.749,4.977,-116.974,-29.559,61.061,-30.609
C05022=1012.749,4.747,-116.955,-29.558,61.051,-30.610
C05023=1012.750,4.515,-116.936,-29.558,61.043,-30.613
C05024=1012.751,4.282,-116.916,-29.558,61.035,-30.616
C05025=1012.751,4.049,-116.896,-29.558,61.026,-30.618
C05026=1012.751,3.821,-116.877,-29.558,61.018,-30.621
C05027=1012.752,3.603,-116.859,-29.558,61.011,-30.623
C05028=1012.752,3.394,-116.841,-29.557,61.004,-30.624
C05029=1012.752,3.003,-116.808,-29.557,60.991,-30.629
C05030=1012.753,2.619,-116.776,-29.558,60.981,-30.634
C05031=1012.753,2.210,-116.741,-29.557,60.969,-30.638
C05032=1012.754,1.990,-116.722,-29.557,60.962,-30.640
C05033=1012.754,1.760,-116.704,-29.557,60.957,-30.641
C05034=1012.754,1.525,-116.684,-29.557,60.950,-30.644
C05035=1012.755,1.289,-116.664,-29.557,60.945,-30.647
C05036=1012.755,1.053,-116.644,-29.557,60.940,-30.648
C05037=1012.755,0.817,-116.624,-29.557,60.934,-30.651
C05038=1012.756,0.582,-116.605,-29.557,60.929,-30.653
C05039=1012.756,0.347,-116.585,-29.558,60.924,-30.657
C05040=1012.757,0.112,-116.565,-29.558,60.919,-30.658
C05041=1012.757,-0.123,-116.545,-29.558,60.914,-30.661
C05042=1012.757,-0.359,-116.525,-29.558,60.910,-30.663
C05043=1012.757,-0.598,-116.505,-29.559,60.906,-30.666
C05044=1012.757,-0.836,-116.486,-29.559,60.903,-30.667
C05045=1012.758,-1.075,-116.465,-29.559,60.898,-30.670
C05046=1012.758,-1.315,-116.445,-29.560,60.895,-30.673
C05047=1012.758,-1.556,-116.425,-29.560,60.892,-30.674
C05048=1012.759,-1.797,-116.404,-29.560,60.889,-30.676
C05049=1012.759,-2.038,-116.384,-29.561,60.886,-30.679
C05050=1012.759,-2.281,-116.364,-29.561,60.883,-30.681
C05051=1012.760,-2.525,-116.343,-29.562,60.881,-30.684
C05052=1012.760,-2.769,-116.323,-29.562,60.879,-30.686
C05053=1012.761,-3.014,-116.302,-29.563,60.877,-30.689
C05054=1012.760,-3.259,-116.282,-29.563,60.875,-30.690
C05055=1012.760,-3.501,-116.261,-29.563,60.874,-30.693
C05056=1012.761,-3.738,-116.241,-29.564,60.873,-30.694
C05057=1012.760,-3.968,-116.222,-29.564,60.873,-30.697
C05058=1012.761,-4.195,-116.203,-29.565,60.871,-30.699
C05059=1012.761,-4.420,-116.184,-29.566,60.871,-30.702
C05060=1012.762,-4.649,-116.164,-29.567,60.871,-30.704
C05061=1012.762,-4.884,-116.145,-29.567,60.870,-30.706
C05062=1012.762,-5.128,-116.125,-29.568,60.872,-30.707
C05063=1012.762,-5.381,-116.103,-29.569,60.871,-30.710
C05064=1012.763,-5.637,-116.082,-29.569,60.872,-30.711
C05065=1012.762,-5.895,-116.060,-29.570,60.873,-30.714
C05066=1012.763,-6.153,-116.038,-29.571,60.875,-30.716
C05067=1012.762,-6.411,-116.016,-29.572,60.876,-30.718
C05068=1012.763,-6.669,-115.994,-29.573,60.878,-30.721
C05069=1012.763,-6.926,-115.973,-29.574,60.880,-30.722
C05070=1012.762,-7.182,-115.952,-29.575,60.882,-30.725
C05071=1012.763,-7.437,-115.930,-29.576,60.885,-30.728
C05072=1012.763,-7.691,-115.908,-29.577,60.888,-30.729
C05073=1012.764,-7.945,-115.887,-29.578,60.890,-30.732
C05074=1012.764,-8.196,-115.866,-29.579,60.894,-30.733
C05075=1012.763,-8.448,-115.845,-29.580,60.898,-30.736
C05076=1012.763,-8.700,-115.824,-29.581,60.902,-30.738
C05077=1012.764,-8.951,-115.803,-29.583,60.906,-30.740
C05078=1012.764,-9.203,-115.782,-29.583,60.911,-30.741
C05079=1012.764,-9.454,-115.761,-29.585,60.915,-30.743
C05080=1012.764,-9.705,-115.739,-29.586,60.920,-30.746
C05081=1012.764,-9.956,-115.718,-29.587,60.925,-30.747
C05082=1012.765,-10.207,-115.697,-29.588,60.930,-30.749
C05083=1012.764,-10.457,-115.677,-29.590,60.936,-30.751
C05084=1012.765,-10.706,-115.655,-29.591,60.942,-30.752
C05085=1012.765,-10.956,-115.634,-29.593,60.948,-30.755
C05086=1012.765,-11.205,-115.613,-29.594,60.954,-30.757
C05087=1012.764,-11.453,-115.592,-29.595,60.960,-30.759
C05088=1012.765,-11.702,-115.571,-29.597,60.968,-30.760
C05089=1012.764,-11.949,-115.551,-29.598,60.974,-30.763
C05090=1012.764,-12.195,-115.530,-29.600,60.982,-30.764
C05091=1012.764,-12.442,-115.510,-29.601,60.990,-30.766
C05092=1012.764,-12.687,-115.489,-29.603,60.997,-30.768
C05093=1012.765,-12.932,-115.468,-29.604,61.005,-30.770
C05094=1012.765,-13.173,-115.448,-29.606,61.013,-30.771
C05095=1012.765,-13.411,-115.428,-29.607,61.022,-30.772
C05096=1012.765,-13.644,-115.409,-29.609,61.030,-30.774
C05097=1012.765,-13.873,-115.389,-29.610,61.038,-30.776
C05098=1012.764,-14.098,-115.370,-29.612,61.047,-30.777
C05099=1012.765,-14.322,-115.352,-29.613,61.055,-30.779
C05100=1012.765,-14.545,-115.332,-29.615,61.063,-30.781
C05101=1012.765,-14.768,-115.314,-29.617,61.073,-30.783
C05102=1012.764,-14.992,-115.295,-29.619,61.083,-30.784
C05103=1012.764,-15.220,-115.276,-29.620,61.092,-30.785
C05104=1012.764,-15.449,-115.257,-29.622,61.103,-30.787
C05105=1012.764,-15.682,-115.237,-29.624,61.113,-30.789
C05106=1012.764,-15.918,-115.218,-29.626,61.124,-30.790
C05107=1012.764,-16.154,-115.197,-29.627,61.134,-30.792
C05108=1012.764,-16.389,-115.177,-29.629,61.145,-30.793
C05109=1012.764,-16.625,-115.158,-29.631,61.157,-30.794
C05110=1012.764,-16.861,-115.138,-29.633,61.169,-30.796
C05111=1012.764,-17.099,-115.118,-29.635,61.181,-30.797
C05112=1012.764,-17.333,-115.098,-29.637,61.193,-30.799
C05113=1012.764,-17.563,-115.079,-29.639,61.205,-30.800
C05114=1012.763,-17.794,-115.059,-29.641,61.217,-30.803
C05115=1012.764,-18.042,-115.039,-29.643,61.231,-30.804
C05116=1012.763,-18.327,-115.014,-29.646,61.246,-30.805
C05117=1012.763,-18.644,-114.988,-29.648,61.264,-30.807
C05118=1012.763,-18.952,-114.962,-29.651,61.283,-30.808
C05119=1012.763,-19.255,-114.937,-29.654,61.300,-30.811
C05120=1012.762,-19.601,-114.908,-29.658,61.321,-30.814
C05121=1012.762,-19.862,-114.886,-29.660,61.338,-30.813
C05122=1012.762,-20.211,-114.856,-29.664,61.360,-30.817
C05123=1012.762,-20.489,-114.834,-29.667,61.378,-30.819
C05124=1012.761,-20.723,-114.813,-29.669,61.393,-30.820
C05125=1012.761,-20.957,-114.794,-29.671,61.409,-30.821
C05126=1012.761,-21.191,-114.774,-29.674,61.425,-30.822
C05127=1012.760,-21.425,-114.754,-29.676,61.441,-30.824
C05128=1012.761,-21.659,-114.734,-29.679,61.457,-30.825
C05129=1012.761,-21.893,-114.715,-29.681,61.474,-30.826
C05130=1012.761,-22.127,-114.695,-29.684,61.490,-30.828
C05131=1012.760,-22.361,-114.675,-29.686,61.508,-30.828
C05132=1012.760,-22.595,-114.656,-29.689,61.526,-30.830
C05133=1012.760,-22.829,-114.636,-29.691,61.543,-30.831
C05134=1012.759,-23.063,-114.617,-29.694,61.561,-30.832
C05135=1012.759,-23.297,-114.597,-29.697,61.579,-30.834
C05136=1012.759,-23.531,-114.577,-29.700,61.597,-30.835
C05137=1012.759,-23.766,-114.558,-29.702,61.615,-30.837
C05138=1012.758,-23.999,-114.538,-29.705,61.635,-30.838
C05139=1012.758,-24.233,-114.518,-29.708,61.653,-30.839
C05140=1012.758,-24.468,-114.499,-29.711,61.673,-30.841
C05141=1012.758,-24.702,-114.479,-29.714,61.692,-30.842
C05142=1012.757,-24.936,-114.459,-29.717,61.712,-30.843
C05143=1012.757,-25.170,-114.439,-29.720,61.732,-30.844
C05144=1012.756,-25.404,-114.420,-29.722,61.752,-30.845
C05145=1012.757,-25.639,-114.400,-29.726,61.772,-30.847
C05146=1012.756,-25.872,-114.380,-29.729,61.793,-30.848
C05147=1012.756,-26.107,-114.361,-29.732,61.814,-30.850
C05148=1012.756,-26.341,-114.341,-29.735,61.835,-30.851
C05149=1012.755,-26.574,-114.321,-29.738,61.857,-30.851
C05150=1012.755,-26.809,-114.302,-29.741,61.879,-30.853
C05151=1012.755,-27.043,-114.282,-29.744,61.900,-30.853
C05152=1012.755,-27.277,-114.263,-29.747,61.922,-30.855
C05153=1012.754,-27.511,-114.243,-29.751,61.945,-30.857
C05154=1012.753,-27.745,-114.223,-29.754,61.968,-30.857
C05155=1012.754,-27.979,-114.204,-29.758,61.991,-30.860
C05156=1012.753,-28.213,-114.184,-29.761,62.014,-30.860
C05157=1012.753,-28.447,-114.164,-29.764,62.037,-30.861
C05158=1012.753,-28.681,-114.145,-29.768,62.061,-30.862
C05159=1012.752,-28.916,-114.125,-29.771,62.085,-30.863
C05160=1012.752,-29.151,-114.105,-29.774,62.109,-30.865
C05161=1012.751,-29.384,-114.085,-29.778,62.133,-30.866
C05162=1012.751,-29.618,-114.066,-29.781,62.158,-30.867
C05163=1012.751,-29.853,-114.046,-29.785,62.183,-30.869
C05164=1012.750,-30.087,-114.027,-29.789,62.208,-30.870
C05165=1012.750,-30.321,-114.006,-29.792,62.234,-30.870
C05166=1012.750,-30.555,-113.987,-29.796,62.258,-30.873
C05167=1012.749,-30.790,-113.967,-29.800,62.284,-30.873
C05168=1012.749,-31.024,-113.948,-29.803,62.311,-30.874
C05169=1012.748,-31.258,-113.928,-29.807,62.337,-30.876
C05170=1012.748,-31.492,-113.908,-29.811,62.363,-30.877
C05171=1012.748,-31.726,-113.889,-29.815,62.391,-30.878
C05172=1012.747,-31.960,-113.869,-29.819,62.418,-30.878
C05173=1012.746,-32.194,-113.849,-29.823,62.445,-30.881
C05174=1012.746,-32.429,-113.829,-29.827,62.473,-30.882
C05175=1012.746,-32.663,-113.810,-29.831,62.500,-30.883
C05176=1012.745,-32.897,-113.790,-29.835,62.528,-30.885
C05177=1012.745,-33.131,-113.770,-29.839,62.557,-30.885
C05178=1012.745,-33.365,-113.751,-29.843,62.585,-30.886
C05179=1012.743,-33.600,-113.731,-29.847,62.615,-30.887
C05180=1012.743,-33.834,-113.711,-29.852,62.643,-30.890
C05181=1012.743,-34.068,-113.692,-29.856,62.672,-30.890
C05182=1012.742,-34.302,-113.672,-29.860,62.702,-30.892
C05183=1012.742,-34.536,-113.652,-29.865,62.732,-30.893
C05184=1012.741,-34.771,-113.632,-29.869,62.762,-30.894
C05185=1012.741,-35.005,-113.613,-29.873,62.792,-30.896
C05186=1012.741,-35.240,-113.593,-29.878,62.823,-30.897
C05187=1012.740,-35.473,-113.573,-29.882,62.853,-30.899
C05188=1012.740,-35.707,-113.554,-29.887,62.885,-30.899
C05189=1012.739,-35.942,-113.534,-29.891,62.917,-30.901
C05190=1012.738,-36.176,-113.514,-29.896,62.948,-30.902
C05191=1012.738,-36.410,-113.494,-29.900,62.980,-30.903
C05192=1012.737,-36.644,-113.475,-29.905,63.012,-30.905
C05193=1012.737,-36.878,-113.455,-29.910,63.044,-30.907
C05194=1012.736,-37.113,-113.435,-29.914,63.077,-30.907
C05195=1012.736,-37.347,-113.416,-29.920,63.109,-30.910
C05196=1012.735,-37.580,-113.396,-29.924,63.142,-30.910
C05197=1012.734,-37.815,-113.377,-29.929,63.176,-30.911
C05198=1012.735,-38.049,-113.357,-29.934,63.210,-30.913
C05199=1012.733,-38.283,-113.337,-29.939,63.243,-30.914
C05200=1012.733,-38.517,-113.317,-29.944,63.278,-30.916
C05201=1012.732,-38.752,-113.298,-29.949,63.312,-30.916
C05202=1012.732,-38.985,-113.278,-29.954,63.346,-30.919
C05203=1012.732,-39.220,-113.258,-29.959,63.382,-30.920
C05204=1012.731,-39.454,-113.239,-29.965,63.416,-30.922
C05205=1012.730,-39.688,-113.219,-29.970,63.452,-30.924
C05206=1012.729,-39.922,-113.199,-29.975,63.487,-30.925
C05207=1012.730,-40.156,-113.180,-29.981,63.524,-30.928
C05208=1012.729,-40.390,-113.160,-29.986,63.560,-30.928
C05209=1012.728,-40.624,-113.140,-29.992,63.597,-30.930
C05210=1012.727,-40.858,-113.120,-29.997,63.633,-30.931
C05211=1012.726,-41.092,-113.101,-30.002,63.669,-30.933
C05212=1012.726,-41.326,-113.081,-30.008,63.707,-30.935
C05213=1012.726,-41.560,-113.061,-30.013,63.744,-30.936
C05214=1012.725,-41.795,-113.042,-30.019,63.782,-30.938
C05215=1012.724,-42.028,-113.022,-30.025,63.820,-30.941
C05216=1012.723,-42.263,-113.002,-30.031,63.858,-30.942
C05217=1012.723,-42.496,-112.982,-30.036,63.896,-30.943
C05218=1012.722,-42.731,-112.963,-30.042,63.935,-30.946
C05219=1012.721,-42.964,-112.943,-30.048,63.974,-30.947
C05220=1012.722,-43.199,-112.923,-30.054,64.014,-30.949
C05221=1012.721,-43.432,-112.903,-30.060,64.053,-30.951
C05222=1012.720,-43.666,-112.884,-30.066,64.093,-30.953
C05223=1012.719,-43.900,-112.864,-30.072,64.132,-30.955
C05224=1012.718,-44.135,-112.845,-30.079,64.172,-30.958
C05225=1012.717,-44.368,-112.825,-30.085,64.213,-30.959
C05226=1012.717,-44.602,-112.805,-30.091,64.254,-30.960
C05227=1012.716,-44.836,-112.785,-30.097,64.294,-30.963
C05228=1012.716,-45.070,-112.766,-30.104,64.336,-30.965
C05229=1012.715,-45.303,-112.746,-30.110,64.378,-30.968
C05230=1012.714,-45.537,-112.726,-30.117,64.420,-30.970
C05231=1012.714,-45.771,-112.707,-30.123,64.462,-30.971
C05232=1012.713,-46.004,-112.687,-30.130,64.504,-30.974
C05233=1012.712,-46.239,-112.668,-30.137,64.546,-30.976
C05234=1012.712,-46.472,-112.647,-30.143,64.589,-30.979
C05235=1012.712,-46.707,-112.628,-30.150,64.632,-30.981
C05236=1012.711,-46.940,-112.608,-30.157,64.676,-30.983
C05237=1012.709,-47.174,-112.588,-30.164,64.719,-30.985
C05238=1012.709,-47.408,-112.569,-30.171,64.762,-30.988
C05239=1012.708,-47.642,-112.549,-30.178,64.807,-30.991
C05240=1012.707,-47.875,-112.529,-30.185,64.852,-30.993
C05241=1012.707,-48.110,-112.509,-30.192,64.897,-30.995
C05242=1012.706,-48.343,-112.490,-30.199,64.941,-30.999
C05243=1012.705,-48.576,-112.470,-30.206,64.986,-31.001
C05244=1012.704,-48.810,-112.451,-30.214,65.031,-31.004
C05245=1012.703,-49.044,-112.431,-30.221,65.076,-31.007
C05246=1012.702,-49.277,-112.411,-30.228,65.123,-31.008
C05247=1012.702,-49.512,-112.392,-30.236,65.169,-31.012
C05248=1012.701,-49.745,-112.372,-30.243,65.215,-31.014
C05249=1012.700,-49.979,-112.352,-30.251,65.262,-31.018
C05250=1012.700,-50.213,-112.333,-30.259,65.309,-31.022
C05251=1012.699,-50.446,-112.313,-30.267,65.356,-31.024
C05252=1012.698,-50.680,-112.293,-30.275,65.403,-31.027
C05253=1012.698,-50.914,-112.273,-30.282,65.450,-31.030
C05254=1012.697,-51.147,-112.254,-30.290,65.499,-31.033
C05255=1012.696,-51.381,-112.234,-30.298,65.547,-31.036
C05256=1012.695,-51.614,-112.214,-30.307,65.596,-31.039
C05257=1012.695,-51.849,-112.194,-30.315,65.645,-31.043
C05258=1012.694,-52.082,-112.174,-30.323,65.694,-31.046
C05259=1012.693,-52.316,-112.154,-30.331,65.743,-31.049
C05260=1012.693,-52.550,-112.135,-30.340,65.793,-31.053
C05261=1012.691,-52.783,-112.116,-30.349,65.842,-31.058
C05262=1012.690,-53.016,-112.096,-30.357,65.893,-31.061
C05263=1012.689,-53.250,-112.076,-30.366,65.943,-31.065
C05264=1012.689,-53.484,-112.057,-30.374,65.993,-31.068
C05265=1012.688,-53.718,-112.037,-30.383,66.044,-31.071
C05266=1012.687,-53.951,-112.017,-30.392,66.095,-31.076
C05267=1012.687,-54.185,-111.997,-30.401,66.147,-31.080
C05268=1012.686,-54.419,-111.978,-30.410,66.198,-31.085
C05269=1012.685,-54.652,-111.958,-30.419,66.250,-31.088
C05270=1012.684,-54.886,-111.938,-30.428,66.301,-31.092
C05271=1012.683,-55.119,-111.918,-30.438,66.354,-31.096
C05272=1012.682,-55.352,-111.898,-30.447,66.407,-31.101
C05273=1012.682,-55.587,-111.879,-30.457,66.460,-31.105
C05274=1012.681,-55.820,-111.859,-30.466,66.513,-31.110
C05275=1012.680,-56.054,-111.839,-30.476,66.566,-31.114
C05276=1012.678,-56.423,-111.808,-30.491,66.652,-31.122
C05277=1012.677,-56.755,-111.780,-30.505,66.728,-31.127
C05278=1012.677,-56.990,-111.761,-30.515,66.784,-31.133
C05279=1012.675,-57.224,-111.740,-30.525,66.838,-31.138
C05280=1012.675,-57.458,-111.721,-30.536,66.894,-31.143
C05281=1012.674,-57.693,-111.701,-30.546,66.948,-31.148
C05282=1012.673,-57.928,-111.681,-30.556,67.004,-31.153
C05283=1012.672,-58.162,-111.661,-30.567,67.060,-31.160
C05284=1012.671,-58.397,-111.641,-30.577,67.117,-31.164
C05285=1012.671,-58.632,-111.621,-30.588,67.174,-31.170
C05286=1012.670,-58.868,-111.602,-30.599,67.230,-31.176
C05287=1012.669,-59.104,-111.582,-30.610,67.288,-31.181
C05288=1012.668,-59.339,-111.561,-30.621,67.345,-31.187
C05289=1012.667,-59.575,-111.542,-30.632,67.404,-31.192
C05290=1012.666,-59.811,-111.522,-30.643,67.462,-31.198
C05291=1012.665,-60.047,-111.502,-30.655,67.521,-31.204
C05292=1012.665,-60.284,-111.482,-30.666,67.579,-31.210
C05293=1012.664,-60.521,-111.462,-30.678,67.639,-31.218
C05294=1012.663,-60.757,-111.442,-30.689,67.698,-31.223
C05295=1012.662,-60.995,-111.422,-30.702,67.758,-31.231
C05296=1012.661,-61.231,-111.402,-30.714,67.818,-31.238
C05297=1012.660,-61.468,-111.382,-30.726,67.878,-31.244
C05298=1012.660,-61.707,-111.361,-30.739,67.939,-31.252
C05299=1012.658,-61.944,-111.341,-30.751,68.001,-31.258
C05300=1012.657,-62.182,-111.321,-30.763,68.062,-31.265
C05301=1012.657,-62.420,-111.301,-30.776,68.123,-31.272
C05302=1012.655,-62.658,-111.281,-30.789,68.186,-31.280
C05303=1012.654,-62.897,-111.261,-30.802,68.248,-31.287
C05304=1012.654,-63.135,-111.240,-30.815,68.311,-31.295
C05305=1012.652,-63.374,-111.220,-30.828,68.373,-31.303
C05306=1012.652,-63.613,-111.201,-30.842,68.437,-31.311
C05307=1012.651,-63.852,-111.180,-30.855,68.500,-31.320
C05308=1012.650,-64.091,-111.160,-30.869,68.564,-31.328
C05309=1012.649,-64.330,-111.139,-30.883,68.628,-31.336
C05310=1012.648,-64.570,-111.119,-30.896,68.693,-31.344
C05311=1012.647,-64.809,-111.099,-30.910,68.757,-31.352
C05312=1012.646,-65.049,-111.078,-30.925,68.822,-31.362
C05313=1012.645,-65.290,-111.058,-30.939,68.888,-31.371
C05314=1012.644,-65.528,-111.038,-30.954,68.954,-31.381
C05315=1012.643,-65.769,-111.018,-30.969,69.020,-31.389
C05316=1012.642,-66.009,-110.998,-30.984,69.086,-31.400
C05317=1012.642,-66.249,-110.977,-30.999,69.153,-31.408
C05318=1012.640,-66.489,-110.956,-31.014,69.220,-31.419
C05319=1012.639,-66.729,-110.936,-31.029,69.287,-31.428
C05320=1012.638,-66.969,-110.916,-31.045,69.355,-31.438
C05321=1012.638,-67.210,-110.895,-31.061,69.423,-31.449
C05322=1012.637,-67.450,-110.875,-31.077,69.491,-31.460
C05323=1012.635,-67.691,-110.855,-31.093,69.559,-31.471
C05324=1012.635,-67.932,-110.834,-31.110,69.627,-31.482
C05325=1012.634,-68.172,-110.814,-31.126,69.696,-31.493
C05326=1012.633,-68.414,-110.793,-31.143,69.766,-31.504
C05327=1012.632,-68.654,-110.773,-31.160,69.835,-31.516
C05328=1012.631,-68.894,-110.753,-31.177,69.905,-31.527
C05329=1012.630,-69.135,-110.732,-31.195,69.975,-31.540
C05330=1012.629,-69.376,-110.712,-31.211,70.045,-31.551
C05331=1012.628,-69.616,-110.691,-31.229,70.115,-31.564
C05332=1012.627,-69.857,-110.671,-31.247,70.186,-31.576
C05333=1012.626,-70.097,-110.650,-31.265,70.257,-31.588
C05334=1012.626,-70.338,-110.631,-31.284,70.329,-31.602
C05335=1012.624,-70.579,-110.610,-31.302,70.401,-31.616
C05336=1012.623,-70.820,-110.589,-31.321,70.472,-31.629
C05337=1012.622,-71.060,-110.569,-31.339,70.544,-31.642
C05338=1012.621,-71.301,-110.548,-31.359,70.618,-31.656
C05339=1012.620,-71.541,-110.528,-31.378,70.689,-31.671
C05340=1012.619,-71.782,-110.508,-31.398,70.763,-31.686
C05341=1012.619,-72.022,-110.487,-31.417,70.835,-31.699
C05342=1012.617,-72.263,-110.467,-31.437,70.910,-31.713
C05343=1012.616,-72.503,-110.447,-31.458,70.984,-31.730
C05344=1012.616,-72.744,-110.426,-31.478,71.058,-31.744
C05345=1012.614,-72.983,-110.405,-31.500,71.132,-31.761
C05346=1012.613,-73.224,-110.385,-31.520,71.206,-31.776
C05347=1012.612,-73.464,-110.365,-31.541,71.280,-31.792
C05348=1012.612,-73.704,-110.344,-31.563,71.355,-31.809
C05349=1012.611,-73.945,-110.324,-31.585,71.432,-31.825
C05350=1012.610,-74.185,-110.304,-31.607,71.506,-31.842
C05351=1012.608,-74.424,-110.283,-31.629,71.583,-31.859
